LIN {X 0,Y 439.387,Z 629.756,A -85,B 0,C 180,E1 -9133.964,E2 -9133.964} C_VEL
LIN {X 0,Y 439.354,Z 629.76,A -85,B 0,C 180,E1 -9136.541,E2 -9136.541} C_VEL
LIN {X 0,Y 439.382,Z 629.757,A -85,B 0,C 180,E1 -9139.019,E2 -9139.019} C_VEL
LIN {X 0,Y 439.376,Z 629.757,A -85,B 0,C 180,E1 -9141.608,E2 -9141.608} C_VEL
LIN {X 0,Y 439.401,Z 629.753,A -85,B 0,C 180,E1 -9144.844,E2 -9144.844} C_VEL
LIN {X 0,Y 439.375,Z 629.756,A -85,B 0,C 180,E1 -9148.14,E2 -9148.14} C_VEL
LIN {X 0,Y 439.434,Z 629.748,A -85,B 0,C 180,E1 -9151.598,E2 -9151.598} C_VEL
LIN {X 0,Y 439.407,Z 629.752,A -85,B 0,C 180,E1 -9154.415,E2 -9154.415} C_VEL
LIN {X 0,Y 439.367,Z 629.759,A -85,B 0,C 180,E1 -9157.425,E2 -9157.425} C_VEL
LIN {X 0,Y 439.443,Z 629.749,A -85,B 0,C 180,E1 -9160.663,E2 -9160.663} C_VEL
LIN {X 0,Y 439.464,Z 629.745,A -85,B 0,C 180,E1 -9164.225,E2 -9164.225} C_VEL
LIN {X 0,Y 439.485,Z 629.743,A -85,B 0,C 180,E1 -9168.001,E2 -9168.001} C_VEL
LIN {X 0,Y 439.55,Z 629.734,A -85,B 0,C 180,E1 -9171.726,E2 -9171.726} C_VEL
LIN {X 0,Y 439.622,Z 629.725,A -85,B 0,C 180,E1 -9174.496,E2 -9174.496} C_VEL
LIN {X 0,Y 439.636,Z 629.724,A -85,B 0,C 180,E1 -9178.168,E2 -9178.168} C_VEL
LIN {X 0,Y 439.765,Z 629.708,A -85,B 0,C 180,E1 -9180,E2 -9180} C_VEL
LIN {X 0,Y 439.658,Z 629.723,A -85,B 0,C 180,E1 -9182.749,E2 -9182.749} C_VEL
LIN {X 0,Y 439.619,Z 629.727,A -85,B 0,C 180,E1 -9186.425,E2 -9186.425} C_VEL
LIN {X 0,Y 439.538,Z 629.738,A -85,B 0,C 180,E1 -9188.274,E2 -9188.274} C_VEL
LIN {X 0,Y 439.466,Z 630.156,A -85,B 0,C 180,E1 -9189.202,E2 -9189.202} C_VEL
LIN {X 0,Y 439.385,Z 633.62,A -85,B 0,C 180,E1 -9192.002,E2 -9192.002} C_VEL
LIN {X 0,Y 439.192,Z 637.24,A -85,B 0,C 180,E1 -9194.835,E2 -9194.835} C_VEL
LIN {X 0,Y 439.017,Z 641.048,A -85,B 0,C 180,E1 -9197.708,E2 -9197.708} C_VEL
LIN {X 0,Y 438.863,Z 644.989,A -85,B 0,C 180,E1 -9200.629,E2 -9200.629} C_VEL
LIN {X 0,Y 438.726,Z 649.729,A -85,B 0,C 180,E1 -9204.064,E2 -9204.064} C_VEL
LIN {X 0,Y 438.588,Z 653.399,A -85,B 0,C 180,E1 -9206.659,E2 -9206.659} C_VEL
LIN {X 0,Y 438.511,Z 656.226,A -85,B 0,C 180,E1 -9208.638,E2 -9208.638} C_VEL
LIN {X 0,Y 441.656,Z 670.395,A -85,B 0,C 180,E1 -9209.231,E2 -9209.231} C_VEL
LIN {X 0,Y 442.692,Z 676.663,A -85,B 0,C 180,E1 -9209.547,E2 -9209.547} C_VEL
LIN {X 0,Y 442.223,Z 688.254,A -85,B 0,C 180,E1 -9210.172,E2 -9210.172} C_VEL
LIN {X 0,Y 441.639,Z 698.968,A -85,B 0,C 180,E1 -9210.92,E2 -9210.92} C_VEL
LIN {X 0,Y 441.047,Z 709.711,A -85,B 0,C 180,E1 -9211.866,E2 -9211.866} C_VEL
LIN {X 0,Y 440.374,Z 720.086,A -85,B 0,C 180,E1 -9212.998,E2 -9212.998} C_VEL
LIN {X 0,Y 439.839,Z 729.502,A -85,B 0,C 180,E1 -9214.281,E2 -9214.281} C_VEL
LIN {X 0,Y 439.34,Z 736.948,A -85,B 0,C 180,E1 -9215.528,E2 -9215.528} C_VEL
LIN {X 0,Y 438.88,Z 744.552,A -85,B 0,C 180,E1 -9217.12,E2 -9217.12} C_VEL
LIN {X 0,Y 438.615,Z 750.268,A -85,B 0,C 180,E1 -9218.675,E2 -9218.675} C_VEL
LIN {X 0,Y 438.473,Z 753.709,A -85,B 0,C 180,E1 -9219.877,E2 -9219.877} C_VEL
LIN {X 0,Y 438.363,Z 756.384,A -85,B 0,C 180,E1 -9221.103,E2 -9221.103} C_VEL
LIN {X 0,Y 438.248,Z 758.479,A -85,B 0,C 180,E1 -9222.465,E2 -9222.465} C_VEL
LIN {X 0,Y 438.176,Z 759.668,A -85,B 0,C 180,E1 -9223.799,E2 -9223.799} C_VEL
LIN {X 0,Y 438.175,Z 760.031,A -85,B 0,C 180,E1 -9225.111,E2 -9225.111} C_VEL
LIN {X 0,Y 438.146,Z 759.584,A -85,B 0,C 180,E1 -9226.391,E2 -9226.391} C_VEL
LIN {X 0,Y 438.226,Z 758.373,A -85,B 0,C 180,E1 -9227.657,E2 -9227.657} C_VEL
LIN {X 0,Y 438.397,Z 755.222,A -85,B 0,C 180,E1 -9229.514,E2 -9229.514} C_VEL
LIN {X 0,Y 438.527,Z 751.961,A -85,B 0,C 180,E1 -9230.81,E2 -9230.81} C_VEL
LIN {X 0,Y 438.792,Z 746.189,A -85,B 0,C 180,E1 -9232.509,E2 -9232.509} C_VEL
LIN {X 0,Y 439.101,Z 739.867,A -85,B 0,C 180,E1 -9233.945,E2 -9233.945} C_VEL
LIN {X 0,Y 439.519,Z 733.401,A -85,B 0,C 180,E1 -9235.134,E2 -9235.134} C_VEL
LIN {X 0,Y 440.041,Z 725.26,A -85,B 0,C 180,E1 -9236.371,E2 -9236.371} C_VEL
LIN {X 0,Y 440.542,Z 716.573,A -85,B 0,C 180,E1 -9237.457,E2 -9237.457} C_VEL
LIN {X 0,Y 441.236,Z 705.818,A -85,B 0,C 180,E1 -9238.54,E2 -9238.54} C_VEL
LIN {X 0,Y 441.75,Z 695.303,A -85,B 0,C 180,E1 -9239.396,E2 -9239.396} C_VEL
LIN {X 0,Y 442.363,Z 683.212,A -85,B 0,C 180,E1 -9240.167,E2 -9240.167} C_VEL
LIN {X 0,Y 442.46,Z 675.311,A -85,B 0,C 180,E1 -9240.567,E2 -9240.567} C_VEL
LIN {X 0,Y 440.025,Z 662.861,A -85,B 0,C 180,E1 -9241.141,E2 -9241.141} C_VEL
LIN {X 0,Y 438.449,Z 655.721,A -85,B 0,C 180,E1 -9241.42,E2 -9241.42} C_VEL
LIN {X 0,Y 438.576,Z 651.43,A -85,B 0,C 180,E1 -9244.363,E2 -9244.363} C_VEL
LIN {X 0,Y 438.669,Z 647.08,A -85,B 0,C 180,E1 -9247.386,E2 -9247.386} C_VEL
LIN {X 0,Y 438.849,Z 642.879,A -85,B 0,C 180,E1 -9250.348,E2 -9250.348} C_VEL
LIN {X 0,Y 439.018,Z 638.03,A -85,B 0,C 180,E1 -9253.845,E2 -9253.845} C_VEL
LIN {X 0,Y 439.064,Z 636.258,A -85,B 0,C 180,E1 -9255.142,E2 -9255.142} C_VEL
LIN {X 0,Y 438.46,Z 635.313,A -85,B 0,C 180,E1 -9255.899,E2 -9255.899} C_VEL
LIN {X 0,Y 435.671,Z 633.985,A -85,B 0,C 180,E1 -9257.135,E2 -9257.135} C_VEL
LIN {X 0,Y 433.291,Z 632.958,A -85,B 0,C 180,E1 -9258.133,E2 -9258.133} C_VEL
LIN {X 0,Y 432.281,Z 632.076,A -85,B 0,C 180,E1 -9258.902,E2 -9258.902} C_VEL
LIN {X 0,Y 432.206,Z 631.749,A -85,B 0,C 180,E1 -9259.162,E2 -9259.162} C_VEL
LIN {X 0,Y 432.239,Z 631.054,A -85,B 0,C 180,E1 -9259.697,E2 -9259.697} C_VEL
LIN {X 0,Y 432.339,Z 630.633,A -85,B 0,C 180,E1 -9260.644,E2 -9260.644} C_VEL
LIN {X 0,Y 432.557,Z 630.605,A -85,B 0,C 180,E1 -9262.531,E2 -9262.531} C_VEL
LIN {X 0,Y 432.6,Z 630.599,A -85,B 0,C 180,E1 -9264.406,E2 -9264.406} C_VEL
LIN {X 0,Y 432.609,Z 630.596,A -85,B 0,C 180,E1 -9268.138,E2 -9268.138} C_VEL
LIN {X 0,Y 432.738,Z 630.58,A -85,B 0,C 180,E1 -9270,E2 -9270} C_VEL
LIN {X 0,Y 432.608,Z 630.6,A -85,B 0,C 180,E1 -9272.793,E2 -9272.793} C_VEL
LIN {X 0,Y 432.556,Z 630.605,A -85,B 0,C 180,E1 -9276.53,E2 -9276.53} C_VEL
LIN {X 0,Y 432.3,Z 630.637,A -85,B 0,C 180,E1 -9279.356,E2 -9279.356} C_VEL
LIN {X 0,Y 431.893,Z 630.707,A -85,B 0,C 180,E1 -9281.736,E2 -9281.736} C_VEL
LIN {X 0,Y 431.726,Z 636.029,A -85,B 0,C 180,E1 -9285.097,E2 -9285.097} C_VEL
LIN {X 0,Y 431.59,Z 640.656,A -85,B 0,C 180,E1 -9288.022,E2 -9288.022} C_VEL
LIN {X 0,Y 431.486,Z 645.367,A -85,B 0,C 180,E1 -9290.997,E2 -9290.997} C_VEL
LIN {X 0,Y 431.407,Z 650.36,A -85,B 0,C 180,E1 -9294.176,E2 -9294.176} C_VEL
LIN {X 0,Y 431.354,Z 655.502,A -85,B 0,C 180,E1 -9297.437,E2 -9297.437} C_VEL
LIN {X 0,Y 434.318,Z 669.166,A -85,B 0,C 180,E1 -9297.986,E2 -9297.986} C_VEL
LIN {X 0,Y 435.698,Z 677.655,A -85,B 0,C 180,E1 -9298.42,E2 -9298.42} C_VEL
LIN {X 0,Y 435.136,Z 689.502,A -85,B 0,C 180,E1 -9299.085,E2 -9299.085} C_VEL
LIN {X 0,Y 434.575,Z 700.253,A -85,B 0,C 180,E1 -9299.867,E2 -9299.867} C_VEL
LIN {X 0,Y 433.897,Z 711.033,A -85,B 0,C 180,E1 -9300.855,E2 -9300.855} C_VEL
LIN {X 0,Y 433.244,Z 721.833,A -85,B 0,C 180,E1 -9302.09,E2 -9302.09} C_VEL
LIN {X 0,Y 432.678,Z 729.989,A -85,B 0,C 180,E1 -9303.243,E2 -9303.243} C_VEL
LIN {X 0,Y 432.171,Z 738.293,A -85,B 0,C 180,E1 -9304.692,E2 -9304.692} C_VEL
LIN {X 0,Y 431.803,Z 745.011,A -85,B 0,C 180,E1 -9306.157,E2 -9306.157} C_VEL
LIN {X 0,Y 431.499,Z 750.36,A -85,B 0,C 180,E1 -9307.644,E2 -9307.644} C_VEL
LIN {X 0,Y 431.308,Z 754.057,A -85,B 0,C 180,E1 -9308.972,E2 -9308.972} C_VEL
LIN {X 0,Y 431.108,Z 757.46,A -85,B 0,C 180,E1 -9310.698,E2 -9310.698} C_VEL
LIN {X 0,Y 431.064,Z 759.055,A -85,B 0,C 180,E1 -9311.947,E2 -9311.947} C_VEL
LIN {X 0,Y 431.022,Z 759.926,A -85,B 0,C 180,E1 -9313.221,E2 -9313.221} C_VEL
LIN {X 0,Y 431.082,Z 760.032,A -85,B 0,C 180,E1 -9314.509,E2 -9314.509} C_VEL
LIN {X 0,Y 431.091,Z 759.371,A -85,B 0,C 180,E1 -9315.833,E2 -9315.833} C_VEL
LIN {X 0,Y 431.14,Z 757.873,A -85,B 0,C 180,E1 -9317.183,E2 -9317.183} C_VEL
LIN {X 0,Y 431.27,Z 755.46,A -85,B 0,C 180,E1 -9318.556,E2 -9318.556} C_VEL
LIN {X 0,Y 431.458,Z 752.01,A -85,B 0,C 180,E1 -9319.958,E2 -9319.958} C_VEL
LIN {X 0,Y 431.725,Z 747.362,A -85,B 0,C 180,E1 -9321.387,E2 -9321.387} C_VEL
LIN {X 0,Y 432.041,Z 740.614,A -85,B 0,C 180,E1 -9322.995,E2 -9322.995} C_VEL
LIN {X 0,Y 432.534,Z 733.555,A -85,B 0,C 180,E1 -9324.332,E2 -9324.332} C_VEL
LIN {X 0,Y 433.12,Z 724.929,A -85,B 0,C 180,E1 -9325.65,E2 -9325.65} C_VEL
LIN {X 0,Y 433.689,Z 715.93,A -85,B 0,C 180,E1 -9326.773,E2 -9326.773} C_VEL
LIN {X 0,Y 434.381,Z 705.148,A -85,B 0,C 180,E1 -9327.866,E2 -9327.866} C_VEL
LIN {X 0,Y 434.999,Z 694.371,A -85,B 0,C 180,E1 -9328.733,E2 -9328.733} C_VEL
LIN {X 0,Y 435.698,Z 681.528,A -85,B 0,C 180,E1 -9329.53,E2 -9329.53} C_VEL
LIN {X 0,Y 435.721,Z 676.839,A -85,B 0,C 180,E1 -9329.772,E2 -9329.772} C_VEL
LIN {X 0,Y 433.464,Z 664.933,A -85,B 0,C 180,E1 -9330.362,E2 -9330.362} C_VEL
LIN {X 0,Y 431.371,Z 655.826,A -85,B 0,C 180,E1 -9330.74,E2 -9330.74} C_VEL
LIN {X 0,Y 431.529,Z 650.765,A -85,B 0,C 180,E1 -9333.913,E2 -9333.913} C_VEL
LIN {X 0,Y 431.533,Z 645.812,A -85,B 0,C 180,E1 -9336.991,E2 -9336.991} C_VEL
LIN {X 0,Y 431.613,Z 640.991,A -85,B 0,C 180,E1 -9340.004,E2 -9340.004} C_VEL
LIN {X 0,Y 431.703,Z 636.112,A -85,B 0,C 180,E1 -9342.96,E2 -9342.96} C_VEL
LIN {X 0,Y 431.894,Z 630.693,A -85,B 0,C 180,E1 -9346.232,E2 -9346.232} C_VEL
LIN {X 0,Y 432.247,Z 630.647,A -85,B 0,C 180,E1 -9348.749,E2 -9348.749} C_VEL
LIN {X 0,Y 432.486,Z 630.616,A -85,B 0,C 180,E1 -9351.59,E2 -9351.59} C_VEL
LIN {X 0,Y 432.595,Z 630.602,A -85,B 0,C 180,E1 -9354.406,E2 -9354.406} C_VEL
LIN {X 0,Y 432.602,Z 630.601,A -85,B 0,C 180,E1 -9358.138,E2 -9358.138} C_VEL
LIN {X 0,Y 432.731,Z 630.585,A -85,B 0,C 180,E1 -9360,E2 -9360} C_VEL
LIN {X 0,Y 432.603,Z 630.6,A -85,B 0,C 180,E1 -9362.794,E2 -9362.794} C_VEL
LIN {X 0,Y 432.569,Z 630.606,A -85,B 0,C 180,E1 -9366.53,E2 -9366.53} C_VEL
LIN {X 0,Y 432.44,Z 630.621,A -85,B 0,C 180,E1 -9369.353,E2 -9369.353} C_VEL
LIN {X 0,Y 432.427,Z 630.623,A -85,B 0,C 180,E1 -9372.804,E2 -9372.804} C_VEL
LIN {X 0,Y 432.409,Z 630.623,A -85,B 0,C 180,E1 -9376.479,E2 -9376.479} C_VEL
LIN {X 0,Y 432.336,Z 630.634,A -85,B 0,C 180,E1 -9379.961,E2 -9379.961} C_VEL
LIN {X 0,Y 432.316,Z 630.636,A -85,B 0,C 180,E1 -9382.964,E2 -9382.964} C_VEL
LIN {X 0,Y 432.361,Z 630.629,A -85,B 0,C 180,E1 -9386.033,E2 -9386.033} C_VEL
LIN {X 0,Y 432.349,Z 630.632,A -85,B 0,C 180,E1 -9389.187,E2 -9389.187} C_VEL
LIN {X 0,Y 432.323,Z 630.636,A -85,B 0,C 180,E1 -9392.294,E2 -9392.294} C_VEL
LIN {X 0,Y 432.338,Z 630.633,A -85,B 0,C 180,E1 -9394.677,E2 -9394.677} C_VEL
LIN {X 0,Y 432.344,Z 630.631,A -85,B 0,C 180,E1 -9398.149,E2 -9398.149} C_VEL
LIN {X 0,Y 432.33,Z 630.633,A -85,B 0,C 180,E1 -9401.603,E2 -9401.603} C_VEL
LIN {X 0,Y 432.331,Z 630.634,A -85,B 0,C 180,E1 -9404.348,E2 -9404.348} C_VEL
LIN {X 0,Y 432.318,Z 630.636,A -85,B 0,C 180,E1 -9407.016,E2 -9407.016} C_VEL
LIN {X 0,Y 432.41,Z 630.692,A -85,B 0,C 180,E1 -9409.809,E2 -9409.809} C_VEL
LIN {X 0,Y 433.314,Z 636.64,A -85,B 0,C 180,E1 -9413.123,E2 -9413.123} C_VEL
LIN {X 0,Y 433.487,Z 641.023,A -85,B 0,C 180,E1 -9415.428,E2 -9415.428} C_VEL
LIN {X 0,Y 433.031,Z 647.602,A -85,B 0,C 180,E1 -9418.712,E2 -9418.712} C_VEL
LIN {X 0,Y 432.656,Z 654.182,A -85,B 0,C 180,E1 -9421.897,E2 -9421.897} C_VEL
LIN {X 0,Y 432.346,Z 660.779,A -85,B 0,C 180,E1 -9424.999,E2 -9424.999} C_VEL
LIN {X 0,Y 432.028,Z 668.48,A -85,B 0,C 180,E1 -9428.53,E2 -9428.53} C_VEL
LIN {X 0,Y 431.751,Z 675.089,A -85,B 0,C 180,E1 -9431.494,E2 -9431.494} C_VEL
LIN {X 0,Y 431.697,Z 679.324,A -85,B 0,C 180,E1 -9433.355,E2 -9433.355} C_VEL
LIN {X 0,Y 433.966,Z 692.719,A -85,B 0,C 180,E1 -9433.836,E2 -9433.836} C_VEL
LIN {X 0,Y 435.473,Z 703.788,A -85,B 0,C 180,E1 -9434.377,E2 -9434.377} C_VEL
LIN {X 0,Y 434.819,Z 716.766,A -85,B 0,C 180,E1 -9435.133,E2 -9435.133} C_VEL
LIN {X 0,Y 434.143,Z 728.744,A -85,B 0,C 180,E1 -9436.048,E2 -9436.048} C_VEL
LIN {X 0,Y 433.519,Z 739.723,A -85,B 0,C 180,E1 -9437.121,E2 -9437.121} C_VEL
LIN {X 0,Y 432.898,Z 749.427,A -85,B 0,C 180,E1 -9438.292,E2 -9438.292} C_VEL
LIN {X 0,Y 432.369,Z 757.388,A -85,B 0,C 180,E1 -9439.464,E2 -9439.464} C_VEL
LIN {X 0,Y 431.913,Z 765.179,A -85,B 0,C 180,E1 -9440.872,E2 -9440.872} C_VEL
LIN {X 0,Y 431.527,Z 772.331,A -85,B 0,C 180,E1 -9442.514,E2 -9442.514} C_VEL
LIN {X 0,Y 431.315,Z 777.274,A -85,B 0,C 180,E1 -9443.98,E2 -9443.98} C_VEL
LIN {X 0,Y 431.283,Z 780.734,A -85,B 0,C 180,E1 -9445.327,E2 -9445.327} C_VEL
LIN {X 0,Y 431.193,Z 782.61,A -85,B 0,C 180,E1 -9446.262,E2 -9446.262} C_VEL
LIN {X 0,Y 431.228,Z 784.02,A -85,B 0,C 180,E1 -9447.198,E2 -9447.198} C_VEL
LIN {X 0,Y 431.199,Z 785.019,A -85,B 0,C 180,E1 -9448.132,E2 -9448.132} C_VEL
LIN {X 0,Y 431.168,Z 785.627,A -85,B 0,C 180,E1 -9449.066,E2 -9449.066} C_VEL
LIN {X 0,Y 431.167,Z 785.842,A -85,B 0,C 180,E1 -9450,E2 -9450} C_VEL
LIN {X 0,Y 431.168,Z 785.62,A -85,B 0,C 180,E1 -9450.934,E2 -9450.934} C_VEL
LIN {X 0,Y 431.199,Z 785.002,A -85,B 0,C 180,E1 -9451.868,E2 -9451.868} C_VEL
LIN {X 0,Y 431.228,Z 783.992,A -85,B 0,C 180,E1 -9452.803,E2 -9452.803} C_VEL
LIN {X 0,Y 431.193,Z 782.577,A -85,B 0,C 180,E1 -9453.738,E2 -9453.738} C_VEL
LIN {X 0,Y 431.316,Z 779.61,A -85,B 0,C 180,E1 -9455.142,E2 -9455.142} C_VEL
LIN {X 0,Y 431.439,Z 775.597,A -85,B 0,C 180,E1 -9456.548,E2 -9456.548} C_VEL
LIN {X 0,Y 431.685,Z 769.429,A -85,B 0,C 180,E1 -9458.19,E2 -9458.19} C_VEL
LIN {X 0,Y 432.03,Z 762.699,A -85,B 0,C 180,E1 -9459.599,E2 -9459.599} C_VEL
LIN {X 0,Y 432.536,Z 754.358,A -85,B 0,C 180,E1 -9461.007,E2 -9461.007} C_VEL
LIN {X 0,Y 433.169,Z 745.811,A -85,B 0,C 180,E1 -9462.177,E2 -9462.177} C_VEL
LIN {X 0,Y 433.695,Z 736.144,A -85,B 0,C 180,E1 -9463.263,E2 -9463.263} C_VEL
LIN {X 0,Y 434.345,Z 724.87,A -85,B 0,C 180,E1 -9464.286,E2 -9464.286} C_VEL
LIN {X 0,Y 435.053,Z 713.507,A -85,B 0,C 180,E1 -9465.099,E2 -9465.099} C_VEL
LIN {X 0,Y 435.436,Z 703.108,A -85,B 0,C 180,E1 -9465.685,E2 -9465.685} C_VEL
LIN {X 0,Y 433.628,Z 689.975,A -85,B 0,C 180,E1 -9466.313,E2 -9466.313} C_VEL
LIN {X 0,Y 431.674,Z 678.73,A -85,B 0,C 180,E1 -9466.737,E2 -9466.737} C_VEL
LIN {X 0,Y 431.916,Z 670.304,A -85,B 0,C 180,E1 -9470.478,E2 -9470.478} C_VEL
LIN {X 0,Y 432.117,Z 663.72,A -85,B 0,C 180,E1 -9473.483,E2 -9473.483} C_VEL
LIN {X 0,Y 432.477,Z 656.969,A -85,B 0,C 180,E1 -9476.647,E2 -9476.647} C_VEL
LIN {X 0,Y 432.876,Z 649.649,A -85,B 0,C 180,E1 -9480.219,E2 -9480.219} C_VEL
LIN {X 0,Y 433.312,Z 643.31,A -85,B 0,C 180,E1 -9483.467,E2 -9483.467} C_VEL
LIN {X 0,Y 433.508,Z 638.901,A -85,B 0,C 180,E1 -9485.845,E2 -9485.845} C_VEL
LIN {X 0,Y 433.084,Z 635.068,A -85,B 0,C 180,E1 -9488.073,E2 -9488.073} C_VEL
LIN {X 0,Y 432.38,Z 630.631,A -85,B 0,C 180,E1 -9490.862,E2 -9490.862} C_VEL
LIN {X 0,Y 432.343,Z 630.634,A -85,B 0,C 180,E1 -9494.346,E2 -9494.346} C_VEL
LIN {X 0,Y 432.322,Z 630.636,A -85,B 0,C 180,E1 -9497.016,E2 -9497.016} C_VEL
LIN {X 0,Y 432.338,Z 630.635,A -85,B 0,C 180,E1 -9499.82,E2 -9499.82} C_VEL
LIN {X 0,Y 432.308,Z 630.637,A -85,B 0,C 180,E1 -9503.022,E2 -9503.022} C_VEL
LIN {X 0,Y 432.361,Z 630.629,A -85,B 0,C 180,E1 -9505.996,E2 -9505.996} C_VEL
LIN {X 0,Y 432.349,Z 630.631,A -85,B 0,C 180,E1 -9509.49,E2 -9509.49} C_VEL
LIN {X 0,Y 432.393,Z 630.626,A -85,B 0,C 180,E1 -9512.928,E2 -9512.928} C_VEL
LIN {X 0,Y 432.373,Z 630.626,A -85,B 0,C 180,E1 -9516.023,E2 -9516.023} C_VEL
LIN {X 0,Y 432.352,Z 630.631,A -85,B 0,C 180,E1 -9519.046,E2 -9519.046} C_VEL
LIN {X 0,Y 432.38,Z 630.628,A -85,B 0,C 180,E1 -9522.011,E2 -9522.011} C_VEL
LIN {X 0,Y 432.397,Z 630.626,A -85,B 0,C 180,E1 -9524.927,E2 -9524.927} C_VEL
LIN {X 0,Y 432.461,Z 630.619,A -85,B 0,C 180,E1 -9527.803,E2 -9527.803} C_VEL
LIN {X 0,Y 432.494,Z 630.614,A -85,B 0,C 180,E1 -9531.59,E2 -9531.59} C_VEL
LIN {X 0,Y 432.599,Z 630.599,A -85,B 0,C 180,E1 -9534.406,E2 -9534.406} C_VEL
LIN {X 0,Y 432.606,Z 630.6,A -85,B 0,C 180,E1 -9538.138,E2 -9538.138} C_VEL
LIN {X 0,Y 432.735,Z 630.584,A -85,B 0,C 180,E1 -9540,E2 -9540} C_VEL
LIN {X 0,Y 432.607,Z 630.601,A -85,B 0,C 180,E1 -9542.794,E2 -9542.794} C_VEL
LIN {X 0,Y 432.574,Z 630.604,A -85,B 0,C 180,E1 -9546.53,E2 -9546.53} C_VEL
LIN {X 0,Y 432.482,Z 630.617,A -85,B 0,C 180,E1 -9548.41,E2 -9548.41} C_VEL
LIN {X 0,Y 432.441,Z 632.519,A -85,B 0,C 180,E1 -9550.298,E2 -9550.298} C_VEL
LIN {X 0,Y 432.234,Z 636.045,A -85,B 0,C 180,E1 -9553.158,E2 -9553.158} C_VEL
LIN {X 0,Y 432.06,Z 640.081,A -85,B 0,C 180,E1 -9556.319,E2 -9556.319} C_VEL
LIN {X 0,Y 431.934,Z 644.029,A -85,B 0,C 180,E1 -9559.314,E2 -9559.314} C_VEL
LIN {X 0,Y 431.672,Z 649.01,A -85,B 0,C 180,E1 -9563.001,E2 -9563.001} C_VEL
LIN {X 0,Y 431.573,Z 653.721,A -85,B 0,C 180,E1 -9566.407,E2 -9566.407} C_VEL
LIN {X 0,Y 431.451,Z 656.452,A -85,B 0,C 180,E1 -9568.348,E2 -9568.348} C_VEL
LIN {X 0,Y 434.724,Z 671.075,A -85,B 0,C 180,E1 -9568.983,E2 -9568.983} C_VEL
LIN {X 0,Y 435.849,Z 678.398,A -85,B 0,C 180,E1 -9569.364,E2 -9569.364} C_VEL
LIN {X 0,Y 435.193,Z 691.24,A -85,B 0,C 180,E1 -9570.108,E2 -9570.108} C_VEL
LIN {X 0,Y 434.561,Z 702.998,A -85,B 0,C 180,E1 -9571.002,E2 -9571.002} C_VEL
LIN {X 0,Y 433.877,Z 713.737,A -85,B 0,C 180,E1 -9572.039,E2 -9572.039} C_VEL
LIN {X 0,Y 433.224,Z 723.639,A -85,B 0,C 180,E1 -9573.228,E2 -9573.228} C_VEL
LIN {X 0,Y 432.747,Z 731.224,A -85,B 0,C 180,E1 -9574.338,E2 -9574.338} C_VEL
LIN {X 0,Y 432.248,Z 738.456,A -85,B 0,C 180,E1 -9575.614,E2 -9575.614} C_VEL
LIN {X 0,Y 431.806,Z 745.281,A -85,B 0,C 180,E1 -9577.106,E2 -9577.106} C_VEL
LIN {X 0,Y 431.559,Z 750.546,A -85,B 0,C 180,E1 -9578.585,E2 -9578.585} C_VEL
LIN {X 0,Y 431.372,Z 754.495,A -85,B 0,C 180,E1 -9580.027,E2 -9580.027} C_VEL
LIN {X 0,Y 431.223,Z 757.315,A -85,B 0,C 180,E1 -9581.435,E2 -9581.435} C_VEL
LIN {X 0,Y 431.094,Z 759.491,A -85,B 0,C 180,E1 -9583.213,E2 -9583.213} C_VEL
LIN {X 0,Y 431.084,Z 760.172,A -85,B 0,C 180,E1 -9584.51,E2 -9584.51} C_VEL
LIN {X 0,Y 431.08,Z 760.092,A -85,B 0,C 180,E1 -9585.836,E2 -9585.836} C_VEL
LIN {X 0,Y 431.092,Z 759.158,A -85,B 0,C 180,E1 -9587.191,E2 -9587.191} C_VEL
LIN {X 0,Y 431.201,Z 757.333,A -85,B 0,C 180,E1 -9588.568,E2 -9588.568} C_VEL
LIN {X 0,Y 431.374,Z 754.534,A -85,B 0,C 180,E1 -9589.972,E2 -9589.972} C_VEL
LIN {X 0,Y 431.531,Z 750.587,A -85,B 0,C 180,E1 -9591.42,E2 -9591.42} C_VEL
LIN {X 0,Y 431.824,Z 745.029,A -85,B 0,C 180,E1 -9592.974,E2 -9592.974} C_VEL
LIN {X 0,Y 432.181,Z 738.493,A -85,B 0,C 180,E1 -9594.399,E2 -9594.399} C_VEL
LIN {X 0,Y 432.748,Z 729.711,A -85,B 0,C 180,E1 -9595.921,E2 -9595.921} C_VEL
LIN {X 0,Y 433.357,Z 720.825,A -85,B 0,C 180,E1 -9597.159,E2 -9597.159} C_VEL
LIN {X 0,Y 433.943,Z 711.272,A -85,B 0,C 180,E1 -9598.24,E2 -9598.24} C_VEL
LIN {X 0,Y 434.627,Z 699.706,A -85,B 0,C 180,E1 -9599.292,E2 -9599.292} C_VEL
LIN {X 0,Y 435.247,Z 688.292,A -85,B 0,C 180,E1 -9600.109,E2 -9600.109} C_VEL
LIN {X 0,Y 435.644,Z 676.629,A -85,B 0,C 180,E1 -9600.751,E2 -9600.751} C_VEL
LIN {X 0,Y 433.236,Z 664.202,A -85,B 0,C 180,E1 -9601.35,E2 -9601.35} C_VEL
LIN {X 0,Y 431.401,Z 655.914,A -85,B 0,C 180,E1 -9601.689,E2 -9601.689} C_VEL
LIN {X 0,Y 431.5,Z 651.224,A -85,B 0,C 180,E1 -9604.946,E2 -9604.946} C_VEL
LIN {X 0,Y 431.652,Z 646.702,A -85,B 0,C 180,E1 -9608.134,E2 -9608.134} C_VEL
LIN {X 0,Y 431.798,Z 642.711,A -85,B 0,C 180,E1 -9611.002,E2 -9611.002} C_VEL
LIN {X 0,Y 431.965,Z 638.68,A -85,B 0,C 180,E1 -9613.943,E2 -9613.943} C_VEL
LIN {X 0,Y 432.191,Z 634.134,A -85,B 0,C 180,E1 -9617.339,E2 -9617.339} C_VEL
LIN {X 0,Y 432.206,Z 631.749,A -85,B 0,C 180,E1 -9619.162,E2 -9619.162} C_VEL
LIN {X 0,Y 431.584,Z 631.102,A -85,B 0,C 180,E1 -9619.934,E2 -9619.934} C_VEL
LIN {X 0,Y 428.862,Z 631.066,A -85,B 0,C 180,E1 -9621.202,E2 -9621.202} C_VEL
LIN {X 0,Y 426.562,Z 631.349,A -85,B 0,C 180,E1 -9622.23,E2 -9622.23} C_VEL
LIN {X 0,Y 425.595,Z 631.473,A -85,B 0,C 180,E1 -9623.023,E2 -9623.023} C_VEL
LIN {X 0,Y 425.527,Z 631.48,A -85,B 0,C 180,E1 -9623.291,E2 -9623.291} C_VEL
LIN {X 0,Y 425.371,Z 631.5,A -85,B 0,C 180,E1 -9625.261,E2 -9625.261} C_VEL
LIN {X 0,Y 425.579,Z 631.471,A -85,B 0,C 180,E1 -9628.107,E2 -9628.107} C_VEL
LIN {X 0,Y 425.707,Z 631.456,A -85,B 0,C 180,E1 -9630,E2 -9630} C_VEL
LIN {X 0,Y 425.559,Z 631.478,A -85,B 0,C 180,E1 -9632.839,E2 -9632.839} C_VEL
LIN {X 0,Y 425.55,Z 631.475,A -85,B 0,C 180,E1 -9635.686,E2 -9635.686} C_VEL
LIN {X 0,Y 425.343,Z 631.504,A -85,B 0,C 180,E1 -9638.552,E2 -9638.552} C_VEL
LIN {X 0,Y 424.936,Z 631.556,A -85,B 0,C 180,E1 -9641.447,E2 -9641.447} C_VEL
LIN {X 0,Y 424.83,Z 631.781,A -85,B 0,C 180,E1 -9641.934,E2 -9641.934} C_VEL
LIN {X 0,Y 424.662,Z 637.169,A -85,B 0,C 180,E1 -9645.354,E2 -9645.354} C_VEL
LIN {X 0,Y 424.515,Z 641.84,A -85,B 0,C 180,E1 -9648.333,E2 -9648.333} C_VEL
LIN {X 0,Y 424.414,Z 647.522,A -85,B 0,C 180,E1 -9651.978,E2 -9651.978} C_VEL
LIN {X 0,Y 424.292,Z 653.067,A -85,B 0,C 180,E1 -9655.509,E2 -9655.509} C_VEL
LIN {X 0,Y 424.269,Z 655.655,A -85,B 0,C 180,E1 -9657.165,E2 -9657.165} C_VEL
LIN {X 0,Y 427.366,Z 669.765,A -85,B 0,C 180,E1 -9657.748,E2 -9657.748} C_VEL
LIN {X 0,Y 428.784,Z 677.926,A -85,B 0,C 180,E1 -9658.18,E2 -9658.18} C_VEL
LIN {X 0,Y 428.249,Z 690.213,A -85,B 0,C 180,E1 -9658.887,E2 -9658.887} C_VEL
LIN {X 0,Y 427.658,Z 700.736,A -85,B 0,C 180,E1 -9659.673,E2 -9659.673} C_VEL
LIN {X 0,Y 426.933,Z 711.53,A -85,B 0,C 180,E1 -9660.684,E2 -9660.684} C_VEL
LIN {X 0,Y 426.292,Z 721.503,A -85,B 0,C 180,E1 -9661.84,E2 -9661.84} C_VEL
LIN {X 0,Y 425.713,Z 729.756,A -85,B 0,C 180,E1 -9663.01,E2 -9663.01} C_VEL
LIN {X 0,Y 425.152,Z 738.171,A -85,B 0,C 180,E1 -9664.488,E2 -9664.488} C_VEL
LIN {X 0,Y 424.786,Z 744.361,A -85,B 0,C 180,E1 -9665.836,E2 -9665.836} C_VEL
LIN {X 0,Y 424.454,Z 749.97,A -85,B 0,C 180,E1 -9667.366,E2 -9667.366} C_VEL
LIN {X 0,Y 424.213,Z 754.514,A -85,B 0,C 180,E1 -9669.016,E2 -9669.016} C_VEL
LIN {X 0,Y 424.037,Z 757.147,A -85,B 0,C 180,E1 -9670.323,E2 -9670.323} C_VEL
LIN {X 0,Y 423.972,Z 759.096,A -85,B 0,C 180,E1 -9671.759,E2 -9671.759} C_VEL
LIN {X 0,Y 423.924,Z 760.093,A -85,B 0,C 180,E1 -9673.159,E2 -9673.159} C_VEL
LIN {X 0,Y 423.984,Z 760.228,A -85,B 0,C 180,E1 -9674.539,E2 -9674.539} C_VEL
LIN {X 0,Y 423.994,Z 759.564,A -85,B 0,C 180,E1 -9675.878,E2 -9675.878} C_VEL
LIN {X 0,Y 424.046,Z 758.147,A -85,B 0,C 180,E1 -9677.194,E2 -9677.194} C_VEL
LIN {X 0,Y 424.18,Z 755.971,A -85,B 0,C 180,E1 -9678.491,E2 -9678.491} C_VEL
LIN {X 0,Y 424.352,Z 753.007,A -85,B 0,C 180,E1 -9679.766,E2 -9679.766} C_VEL
LIN {X 0,Y 424.634,Z 748.084,A -85,B 0,C 180,E1 -9681.375,E2 -9681.375} C_VEL
LIN {X 0,Y 424.997,Z 741.412,A -85,B 0,C 180,E1 -9683.019,E2 -9683.019} C_VEL
LIN {X 0,Y 425.494,Z 734.476,A -85,B 0,C 180,E1 -9684.378,E2 -9684.378} C_VEL
LIN {X 0,Y 426.106,Z 725.939,A -85,B 0,C 180,E1 -9685.736,E2 -9685.736} C_VEL
LIN {X 0,Y 426.728,Z 716.57,A -85,B 0,C 180,E1 -9686.937,E2 -9686.937} C_VEL
LIN {X 0,Y 427.448,Z 706.609,A -85,B 0,C 180,E1 -9687.978,E2 -9687.978} C_VEL
LIN {X 0,Y 428.096,Z 695.689,A -85,B 0,C 180,E1 -9688.9,E2 -9688.9} C_VEL
LIN {X 0,Y 428.767,Z 683.987,A -85,B 0,C 180,E1 -9689.665,E2 -9689.665} C_VEL
LIN {X 0,Y 428.856,Z 677.61,A -85,B 0,C 180,E1 -9690.011,E2 -9690.011} C_VEL
LIN {X 0,Y 426.364,Z 664.772,A -85,B 0,C 180,E1 -9690.668,E2 -9690.668} C_VEL
LIN {X 0,Y 424.308,Z 656.041,A -85,B 0,C 180,E1 -9691.021,E2 -9691.021} C_VEL
LIN {X 0,Y 424.436,Z 650.526,A -85,B 0,C 180,E1 -9694.499,E2 -9694.499} C_VEL
LIN {X 0,Y 424.502,Z 644.97,A -85,B 0,C 180,E1 -9697.99,E2 -9697.99} C_VEL
LIN {X 0,Y 424.619,Z 640.631,A -85,B 0,C 180,E1 -9700.669,E2 -9700.669} C_VEL
LIN {X 0,Y 424.69,Z 635.637,A -85,B 0,C 180,E1 -9703.699,E2 -9703.699} C_VEL
LIN {X 0,Y 424.852,Z 631.57,A -85,B 0,C 180,E1 -9706.121,E2 -9706.121} C_VEL
LIN {X 0,Y 425.187,Z 631.526,A -85,B 0,C 180,E1 -9708.559,E2 -9708.559} C_VEL
LIN {X 0,Y 425.435,Z 631.495,A -85,B 0,C 180,E1 -9711.45,E2 -9711.45} C_VEL
LIN {X 0,Y 425.551,Z 631.48,A -85,B 0,C 180,E1 -9714.313,E2 -9714.313} C_VEL
LIN {X 0,Y 425.572,Z 631.477,A -85,B 0,C 180,E1 -9718.107,E2 -9718.107} C_VEL
LIN {X 0,Y 425.701,Z 631.46,A -85,B 0,C 180,E1 -9720,E2 -9720} C_VEL
LIN {X 0,Y 425.554,Z 631.478,A -85,B 0,C 180,E1 -9722.84,E2 -9722.84} C_VEL
LIN {X 0,Y 425.527,Z 631.482,A -85,B 0,C 180,E1 -9726.639,E2 -9726.639} C_VEL
LIN {X 0,Y 425.399,Z 631.497,A -85,B 0,C 180,E1 -9729.509,E2 -9729.509} C_VEL
LIN {X 0,Y 425.389,Z 631.499,A -85,B 0,C 180,E1 -9732.904,E2 -9732.904} C_VEL
LIN {X 0,Y 425.358,Z 631.502,A -85,B 0,C 180,E1 -9736.605,E2 -9736.605} C_VEL
LIN {X 0,Y 425.325,Z 631.506,A -85,B 0,C 180,E1 -9739.636,E2 -9739.636} C_VEL
LIN {X 0,Y 425.303,Z 631.508,A -85,B 0,C 180,E1 -9743.365,E2 -9743.365} C_VEL
LIN {X 0,Y 425.345,Z 631.503,A -85,B 0,C 180,E1 -9746.845,E2 -9746.845} C_VEL
LIN {X 0,Y 425.315,Z 631.508,A -85,B 0,C 180,E1 -9749.718,E2 -9749.718} C_VEL
LIN {X 0,Y 425.279,Z 631.512,A -85,B 0,C 180,E1 -9753.048,E2 -9753.048} C_VEL
LIN {X 0,Y 425.282,Z 631.511,A -85,B 0,C 180,E1 -9755.93,E2 -9755.93} C_VEL
LIN {X 0,Y 425.298,Z 631.51,A -85,B 0,C 180,E1 -9759.044,E2 -9759.044} C_VEL
LIN {X 0,Y 425.272,Z 631.514,A -85,B 0,C 180,E1 -9762.654,E2 -9762.654} C_VEL
LIN {X 0,Y 425.259,Z 631.515,A -85,B 0,C 180,E1 -9766.045,E2 -9766.045} C_VEL
LIN {X 0,Y 425.319,Z 631.515,A -85,B 0,C 180,E1 -9769.553,E2 -9769.553} C_VEL
LIN {X 0,Y 426.135,Z 636.492,A -85,B 0,C 180,E1 -9772.395,E2 -9772.395} C_VEL
LIN {X 0,Y 426.51,Z 640.877,A -85,B 0,C 180,E1 -9774.78,E2 -9774.78} C_VEL
LIN {X 0,Y 426.085,Z 647.443,A -85,B 0,C 180,E1 -9778.142,E2 -9778.142} C_VEL
LIN {X 0,Y 425.693,Z 654.008,A -85,B 0,C 180,E1 -9781.395,E2 -9781.395} C_VEL
LIN {X 0,Y 425.318,Z 660.596,A -85,B 0,C 180,E1 -9784.557,E2 -9784.557} C_VEL
LIN {X 0,Y 425.031,Z 667.563,A -85,B 0,C 180,E1 -9787.816,E2 -9787.816} C_VEL
LIN {X 0,Y 424.698,Z 674.878,A -85,B 0,C 180,E1 -9791.175,E2 -9791.175} C_VEL
LIN {X 0,Y 424.626,Z 679.046,A -85,B 0,C 180,E1 -9793.059,E2 -9793.059} C_VEL
LIN {X 0,Y 427.211,Z 694.635,A -85,B 0,C 180,E1 -9793.671,E2 -9793.671} C_VEL
LIN {X 0,Y 428.515,Z 705.594,A -85,B 0,C 180,E1 -9794.239,E2 -9794.239} C_VEL
LIN {X 0,Y 427.843,Z 718.128,A -85,B 0,C 180,E1 -9795.006,E2 -9795.006} C_VEL
LIN {X 0,Y 427.143,Z 729.533,A -85,B 0,C 180,E1 -9795.921,E2 -9795.921} C_VEL
LIN {X 0,Y 426.483,Z 740.471,A -85,B 0,C 180,E1 -9797.025,E2 -9797.025} C_VEL
LIN {X 0,Y 425.893,Z 749.122,A -85,B 0,C 180,E1 -9798.096,E2 -9798.096} C_VEL
LIN {X 0,Y 425.336,Z 757.1,A -85,B 0,C 180,E1 -9799.288,E2 -9799.288} C_VEL
LIN {X 0,Y 424.858,Z 764.912,A -85,B 0,C 180,E1 -9800.719,E2 -9800.719} C_VEL
LIN {X 0,Y 424.558,Z 770.238,A -85,B 0,C 180,E1 -9801.912,E2 -9801.912} C_VEL
LIN {X 0,Y 424.259,Z 776.436,A -85,B 0,C 180,E1 -9803.681,E2 -9803.681} C_VEL
LIN {X 0,Y 424.213,Z 780.503,A -85,B 0,C 180,E1 -9805.249,E2 -9805.249} C_VEL
LIN {X 0,Y 424.105,Z 782.384,A -85,B 0,C 180,E1 -9806.2,E2 -9806.2} C_VEL
LIN {X 0,Y 424.125,Z 783.799,A -85,B 0,C 180,E1 -9807.151,E2 -9807.151} C_VEL
LIN {X 0,Y 424.125,Z 784.803,A -85,B 0,C 180,E1 -9808.101,E2 -9808.101} C_VEL
LIN {X 0,Y 424.084,Z 785.631,A -85,B 0,C 180,E1 -9810,E2 -9810} C_VEL
LIN {X 0,Y 424.088,Z 785.413,A -85,B 0,C 180,E1 -9810.95,E2 -9810.95} C_VEL
LIN {X 0,Y 424.125,Z 784.797,A -85,B 0,C 180,E1 -9811.9,E2 -9811.9} C_VEL
LIN {X 0,Y 424.125,Z 783.788,A -85,B 0,C 180,E1 -9812.85,E2 -9812.85} C_VEL
LIN {X 0,Y 424.105,Z 782.375,A -85,B 0,C 180,E1 -9813.801,E2 -9813.801} C_VEL
LIN {X 0,Y 424.23,Z 779.409,A -85,B 0,C 180,E1 -9815.228,E2 -9815.228} C_VEL
LIN {X 0,Y 424.354,Z 775.397,A -85,B 0,C 180,E1 -9816.658,E2 -9816.658} C_VEL
LIN {X 0,Y 424.619,Z 769.234,A -85,B 0,C 180,E1 -9818.327,E2 -9818.327} C_VEL
LIN {X 0,Y 425,Z 762.505,A -85,B 0,C 180,E1 -9819.759,E2 -9819.759} C_VEL
LIN {X 0,Y 425.519,Z 754.166,A -85,B 0,C 180,E1 -9821.191,E2 -9821.191} C_VEL
LIN {X 0,Y 426.205,Z 745.627,A -85,B 0,C 180,E1 -9822.379,E2 -9822.379} C_VEL
LIN {X 0,Y 426.812,Z 735.336,A -85,B 0,C 180,E1 -9823.546,E2 -9823.546} C_VEL
LIN {X 0,Y 427.442,Z 724.71,A -85,B 0,C 180,E1 -9824.522,E2 -9824.522} C_VEL
LIN {X 0,Y 428.175,Z 713.391,A -85,B 0,C 180,E1 -9825.348,E2 -9825.348} C_VEL
LIN {X 0,Y 428.571,Z 704.164,A -85,B 0,C 180,E1 -9825.882,E2 -9825.882} C_VEL
LIN {X 0,Y 426.767,Z 690.673,A -85,B 0,C 180,E1 -9826.564,E2 -9826.564} C_VEL
LIN {X 0,Y 424.617,Z 678.562,A -85,B 0,C 180,E1 -9827.02,E2 -9827.02} C_VEL
LIN {X 0,Y 424.889,Z 670.148,A -85,B 0,C 180,E1 -9830.832,E2 -9830.832} C_VEL
LIN {X 0,Y 425.111,Z 663.586,A -85,B 0,C 180,E1 -9833.894,E2 -9833.894} C_VEL
LIN {X 0,Y 425.443,Z 657.379,A -85,B 0,C 180,E1 -9836.869,E2 -9836.869} C_VEL
LIN {X 0,Y 425.842,Z 650.643,A -85,B 0,C 180,E1 -9840.223,E2 -9840.223} C_VEL
LIN {X 0,Y 426.311,Z 644.319,A -85,B 0,C 180,E1 -9843.523,E2 -9843.523} C_VEL
LIN {X 0,Y 426.521,Z 641.219,A -85,B 0,C 180,E1 -9845.22,E2 -9845.22} C_VEL
LIN {X 0,Y 426.201,Z 637.003,A -85,B 0,C 180,E1 -9847.673,E2 -9847.673} C_VEL
LIN {X 0,Y 425.493,Z 632.453,A -85,B 0,C 180,E1 -9850.554,E2 -9850.554} C_VEL
LIN {X 0,Y 425.313,Z 631.511,A -85,B 0,C 180,E1 -9851.261,E2 -9851.261} C_VEL
LIN {X 0,Y 425.291,Z 631.511,A -85,B 0,C 180,E1 -9854.718,E2 -9854.718} C_VEL
LIN {X 0,Y 425.292,Z 631.512,A -85,B 0,C 180,E1 -9858.042,E2 -9858.042} C_VEL
LIN {X 0,Y 425.309,Z 631.511,A -85,B 0,C 180,E1 -9861.102,E2 -9861.102} C_VEL
LIN {X 0,Y 425.301,Z 631.51,A -85,B 0,C 180,E1 -9864.664,E2 -9864.664} C_VEL
LIN {X 0,Y 425.267,Z 631.513,A -85,B 0,C 180,E1 -9868.073,E2 -9868.073} C_VEL
LIN {X 0,Y 425.333,Z 631.505,A -85,B 0,C 180,E1 -9871.368,E2 -9871.368} C_VEL
LIN {X 0,Y 425.297,Z 631.511,A -85,B 0,C 180,E1 -9874.555,E2 -9874.555} C_VEL
LIN {X 0,Y 425.289,Z 631.511,A -85,B 0,C 180,E1 -9877.661,E2 -9877.661} C_VEL
LIN {X 0,Y 425.364,Z 631.503,A -85,B 0,C 180,E1 -9880.704,E2 -9880.704} C_VEL
LIN {X 0,Y 425.39,Z 631.499,A -85,B 0,C 180,E1 -9883.688,E2 -9883.688} C_VEL
LIN {X 0,Y 425.414,Z 631.496,A -85,B 0,C 180,E1 -9887.598,E2 -9887.598} C_VEL
LIN {X 0,Y 425.444,Z 631.493,A -85,B 0,C 180,E1 -9891.45,E2 -9891.45} C_VEL
LIN {X 0,Y 425.556,Z 631.477,A -85,B 0,C 180,E1 -9894.313,E2 -9894.313} C_VEL
LIN {X 0,Y 425.575,Z 631.476,A -85,B 0,C 180,E1 -9898.107,E2 -9898.107} C_VEL
LIN {X 0,Y 425.705,Z 631.46,A -85,B 0,C 180,E1 -9900,E2 -9900} C_VEL
LIN {X 0,Y 425.559,Z 631.479,A -85,B 0,C 180,E1 -9902.84,E2 -9902.84} C_VEL
LIN {X 0,Y 425.531,Z 631.482,A -85,B 0,C 180,E1 -9906.639,E2 -9906.639} C_VEL
LIN {X 0,Y 425.421,Z 631.501,A -85,B 0,C 180,E1 -9908.551,E2 -9908.551} C_VEL
LIN {X 0,Y 425.322,Z 634.917,A -85,B 0,C 180,E1 -9911.437,E2 -9911.437} C_VEL
LIN {X 0,Y 425.126,Z 638.495,A -85,B 0,C 180,E1 -9914.358,E2 -9914.358} C_VEL
LIN {X 0,Y 424.933,Z 642.278,A -85,B 0,C 180,E1 -9917.32,E2 -9917.32} C_VEL
LIN {X 0,Y 424.761,Z 646.215,A -85,B 0,C 180,E1 -9920.332,E2 -9920.332} C_VEL
LIN {X 0,Y 424.597,Z 650.311,A -85,B 0,C 180,E1 -9923.407,E2 -9923.407} C_VEL
LIN {X 0,Y 424.478,Z 654.692,A -85,B 0,C 180,E1 -9926.611,E2 -9926.611} C_VEL
LIN {X 0,Y 424.404,Z 656.887,A -85,B 0,C 180,E1 -9928.06,E2 -9928.06} C_VEL
LIN {X 0,Y 427.424,Z 669.755,A -85,B 0,C 180,E1 -9928.621,E2 -9928.621} C_VEL
LIN {X 0,Y 429.021,Z 678.909,A -85,B 0,C 180,E1 -9929.112,E2 -9929.112} C_VEL
LIN {X 0,Y 428.366,Z 691.633,A -85,B 0,C 180,E1 -9929.867,E2 -9929.867} C_VEL
LIN {X 0,Y 427.736,Z 702.77,A -85,B 0,C 180,E1 -9930.726,E2 -9930.726} C_VEL
LIN {X 0,Y 426.997,Z 713.635,A -85,B 0,C 180,E1 -9931.782,E2 -9931.782} C_VEL
LIN {X 0,Y 426.295,Z 723.361,A -85,B 0,C 180,E1 -9932.96,E2 -9932.96} C_VEL
LIN {X 0,Y 425.681,Z 732.719,A -85,B 0,C 180,E1 -9934.361,E2 -9934.361} C_VEL
LIN {X 0,Y 425.087,Z 740.815,A -85,B 0,C 180,E1 -9935.892,E2 -9935.892} C_VEL
LIN {X 0,Y 424.683,Z 747.155,A -85,B 0,C 180,E1 -9937.407,E2 -9937.407} C_VEL
LIN {X 0,Y 424.434,Z 752.314,A -85,B 0,C 180,E1 -9938.993,E2 -9938.993} C_VEL
LIN {X 0,Y 424.2,Z 756.703,A -85,B 0,C 180,E1 -9940.899,E2 -9940.899} C_VEL
LIN {X 0,Y 424.092,Z 758.15,A -85,B 0,C 180,E1 -9941.778,E2 -9941.778} C_VEL
LIN {X 0,Y 424.001,Z 759.701,A -85,B 0,C 180,E1 -9943.17,E2 -9943.17} C_VEL
LIN {X 0,Y 423.986,Z 760.391,A -85,B 0,C 180,E1 -9944.539,E2 -9944.539} C_VEL
LIN {X 0,Y 423.98,Z 760.285,A -85,B 0,C 180,E1 -9945.877,E2 -9945.877} C_VEL
LIN {X 0,Y 423.995,Z 759.393,A -85,B 0,C 180,E1 -9947.187,E2 -9947.187} C_VEL
LIN {X 0,Y 424.115,Z 757.745,A -85,B 0,C 180,E1 -9948.483,E2 -9948.483} C_VEL
LIN {X 0,Y 424.274,Z 755.383,A -85,B 0,C 180,E1 -9949.757,E2 -9949.757} C_VEL
LIN {X 0,Y 424.405,Z 752.019,A -85,B 0,C 180,E1 -9951.106,E2 -9951.106} C_VEL
LIN {X 0,Y 424.675,Z 747.135,A -85,B 0,C 180,E1 -9952.595,E2 -9952.595} C_VEL
LIN {X 0,Y 425.02,Z 740.734,A -85,B 0,C 180,E1 -9954.121,E2 -9954.121} C_VEL
LIN {X 0,Y 425.558,Z 732.559,A -85,B 0,C 180,E1 -9955.664,E2 -9955.664} C_VEL
LIN {X 0,Y 426.229,Z 723.373,A -85,B 0,C 180,E1 -9957.035,E2 -9957.035} C_VEL
LIN {X 0,Y 426.893,Z 713.677,A -85,B 0,C 180,E1 -9958.209,E2 -9958.209} C_VEL
LIN {X 0,Y 427.574,Z 702.873,A -85,B 0,C 180,E1 -9959.264,E2 -9959.264} C_VEL
LIN {X 0,Y 428.2,Z 691.606,A -85,B 0,C 180,E1 -9960.134,E2 -9960.134} C_VEL
LIN {X 0,Y 428.872,Z 679.153,A -85,B 0,C 180,E1 -9960.874,E2 -9960.874} C_VEL
LIN {X 0,Y 427.154,Z 668.955,A -85,B 0,C 180,E1 -9961.409,E2 -9961.409} C_VEL
LIN {X 0,Y 424.331,Z 656.082,A -85,B 0,C 180,E1 -9961.968,E2 -9961.968} C_VEL
LIN {X 0,Y 424.432,Z 652.486,A -85,B 0,C 180,E1 -9964.499,E2 -9964.499} C_VEL
LIN {X 0,Y 424.578,Z 647.626,A -85,B 0,C 180,E1 -9967.967,E2 -9967.967} C_VEL
LIN {X 0,Y 424.728,Z 643.893,A -85,B 0,C 180,E1 -9970.674,E2 -9970.674} C_VEL
LIN {X 0,Y 424.899,Z 639.838,A -85,B 0,C 180,E1 -9973.669,E2 -9973.669} C_VEL
LIN {X 0,Y 425.154,Z 635.113,A -85,B 0,C 180,E1 -9977.24,E2 -9977.24} C_VEL
LIN {X 0,Y 425.184,Z 632.162,A -85,B 0,C 180,E1 -9979.524,E2 -9979.524} C_VEL
LIN {X 0,Y 425.261,Z 631.514,A -85,B 0,C 180,E1 -9980.487,E2 -9980.487} C_VEL
LIN {X 0,Y 425.541,Z 631.477,A -85,B 0,C 180,E1 -9982.407,E2 -9982.407} C_VEL
LIN {X 0,Y 425.527,Z 631.48,A -85,B 0,C 180,E1 -9983.291,E2 -9983.291} C_VEL
LIN {X 0,Y 424.887,Z 631.565,A -85,B 0,C 180,E1 -9984.079,E2 -9984.079} C_VEL
LIN {X 0,Y 422.038,Z 631.923,A -85,B 0,C 180,E1 -9985.36,E2 -9985.36} C_VEL
LIN {X 0,Y 419.617,Z 632.221,A -85,B 0,C 180,E1 -9986.394,E2 -9986.394} C_VEL
LIN {X 0,Y 418.589,Z 632.345,A -85,B 0,C 180,E1 -9987.193,E2 -9987.193} C_VEL
LIN {X 0,Y 418.512,Z 632.352,A -85,B 0,C 180,E1 -9987.464,E2 -9987.464} C_VEL
LIN {X 0,Y 418.677,Z 632.331,A -85,B 0,C 180,E1 -9990,E2 -9990} C_VEL
LIN {X 0,Y 418.513,Z 632.356,A -85,B 0,C 180,E1 -9992.887,E2 -9992.887} C_VEL
LIN {X 0,Y 418.508,Z 632.352,A -85,B 0,C 180,E1 -9995.782,E2 -9995.782} C_VEL
LIN {X 0,Y 418.271,Z 632.386,A -85,B 0,C 180,E1 -9998.697,E2 -9998.697} C_VEL
LIN {X 0,Y 417.807,Z 632.443,A -85,B 0,C 180,E1 -10001.763,E2 -10001.763} C_VEL
LIN {X 0,Y 417.594,Z 638.307,A -85,B 0,C 180,E1 -10005.621,E2 -10005.621} C_VEL
LIN {X 0,Y 417.459,Z 643.024,A -85,B 0,C 180,E1 -10008.654,E2 -10008.654} C_VEL
LIN {X 0,Y 417.32,Z 648.438,A -85,B 0,C 180,E1 -10012.143,E2 -10012.143} C_VEL
LIN {X 0,Y 417.244,Z 652.723,A -85,B 0,C 180,E1 -10014.903,E2 -10014.903} C_VEL
LIN {X 0,Y 417.221,Z 655.949,A -85,B 0,C 180,E1 -10016.899,E2 -10016.899} C_VEL
LIN {X 0,Y 420.273,Z 669.775,A -85,B 0,C 180,E1 -10017.472,E2 -10017.472} C_VEL
LIN {X 0,Y 421.919,Z 679.749,A -85,B 0,C 180,E1 -10018.014,E2 -10018.014} C_VEL
LIN {X 0,Y 421.273,Z 692.301,A -85,B 0,C 180,E1 -10018.783,E2 -10018.783} C_VEL
LIN {X 0,Y 420.531,Z 704.452,A -85,B 0,C 180,E1 -10019.757,E2 -10019.757} C_VEL
LIN {X 0,Y 419.771,Z 715.11,A -85,B 0,C 180,E1 -10020.846,E2 -10020.846} C_VEL
LIN {X 0,Y 419.028,Z 725.533,A -85,B 0,C 180,E1 -10022.175,E2 -10022.175} C_VEL
LIN {X 0,Y 418.458,Z 733.688,A -85,B 0,C 180,E1 -10023.461,E2 -10023.461} C_VEL
LIN {X 0,Y 417.984,Z 740.899,A -85,B 0,C 180,E1 -10024.867,E2 -10024.867} C_VEL
LIN {X 0,Y 417.585,Z 747.163,A -85,B 0,C 180,E1 -10026.387,E2 -10026.387} C_VEL
LIN {X 0,Y 417.278,Z 752.551,A -85,B 0,C 180,E1 -10028.076,E2 -10028.076} C_VEL
LIN {X 0,Y 417.002,Z 756.527,A -85,B 0,C 180,E1 -10029.824,E2 -10029.824} C_VEL
LIN {X 0,Y 416.887,Z 758.57,A -85,B 0,C 180,E1 -10031.107,E2 -10031.107} C_VEL
LIN {X 0,Y 416.855,Z 759.868,A -85,B 0,C 180,E1 -10032.405,E2 -10032.405} C_VEL
LIN {X 0,Y 416.85,Z 760.44,A -85,B 0,C 180,E1 -10033.728,E2 -10033.728} C_VEL
LIN {X 0,Y 416.892,Z 760.269,A -85,B 0,C 180,E1 -10035.075,E2 -10035.075} C_VEL
LIN {X 0,Y 416.915,Z 759.298,A -85,B 0,C 180,E1 -10036.456,E2 -10036.456} C_VEL
LIN {X 0,Y 417.072,Z 756.498,A -85,B 0,C 180,E1 -10038.394,E2 -10038.394} C_VEL
LIN {X 0,Y 417.261,Z 753.502,A -85,B 0,C 180,E1 -10039.753,E2 -10039.753} C_VEL
LIN {X 0,Y 417.574,Z 748.36,A -85,B 0,C 180,E1 -10041.484,E2 -10041.484} C_VEL
LIN {X 0,Y 417.934,Z 742.344,A -85,B 0,C 180,E1 -10043.016,E2 -10043.016} C_VEL
LIN {X 0,Y 418.506,Z 734.5,A -85,B 0,C 180,E1 -10044.594,E2 -10044.594} C_VEL
LIN {X 0,Y 419.188,Z 725.905,A -85,B 0,C 180,E1 -10045.975,E2 -10045.975} C_VEL
LIN {X 0,Y 419.876,Z 716.265,A -85,B 0,C 180,E1 -10047.223,E2 -10047.223} C_VEL
LIN {X 0,Y 420.602,Z 705.817,A -85,B 0,C 180,E1 -10048.32,E2 -10048.32} C_VEL
LIN {X 0,Y 421.379,Z 694.142,A -85,B 0,C 180,E1 -10049.284,E2 -10049.284} C_VEL
LIN {X 0,Y 422.062,Z 682.514,A -85,B 0,C 180,E1 -10050.03,E2 -10050.03} C_VEL
LIN {X 0,Y 421.907,Z 677.83,A -85,B 0,C 180,E1 -10050.293,E2 -10050.293} C_VEL
LIN {X 0,Y 419.512,Z 665.695,A -85,B 0,C 180,E1 -10050.933,E2 -10050.933} C_VEL
LIN {X 0,Y 417.251,Z 656.186,A -85,B 0,C 180,E1 -10051.348,E2 -10051.348} C_VEL
LIN {X 0,Y 417.346,Z 651.983,A -85,B 0,C 180,E1 -10054.034,E2 -10054.034} C_VEL
LIN {X 0,Y 417.437,Z 645.983,A -85,B 0,C 180,E1 -10057.815,E2 -10057.815} C_VEL
LIN {X 0,Y 417.555,Z 640.394,A -85,B 0,C 180,E1 -10061.349,E2 -10061.349} C_VEL
LIN {X 0,Y 417.676,Z 635.415,A -85,B 0,C 180,E1 -10064.382,E2 -10064.382} C_VEL
LIN {X 0,Y 417.778,Z 632.452,A -85,B 0,C 180,E1 -10066.13,E2 -10066.13} C_VEL
LIN {X 0,Y 418.13,Z 632.405,A -85,B 0,C 180,E1 -10068.364,E2 -10068.364} C_VEL
LIN {X 0,Y 418.391,Z 632.372,A -85,B 0,C 180,E1 -10071.305,E2 -10071.305} C_VEL
LIN {X 0,Y 418.51,Z 632.358,A -85,B 0,C 180,E1 -10074.217,E2 -10074.217} C_VEL
LIN {X 0,Y 418.541,Z 632.352,A -85,B 0,C 180,E1 -10078.075,E2 -10078.075} C_VEL
LIN {X 0,Y 418.671,Z 632.336,A -85,B 0,C 180,E1 -10080,E2 -10080} C_VEL
LIN {X 0,Y 418.508,Z 632.356,A -85,B 0,C 180,E1 -10082.888,E2 -10082.888} C_VEL
LIN {X 0,Y 418.49,Z 632.358,A -85,B 0,C 180,E1 -10086.751,E2 -10086.751} C_VEL
LIN {X 0,Y 418.339,Z 632.376,A -85,B 0,C 180,E1 -10089.671,E2 -10089.671} C_VEL
LIN {X 0,Y 418.342,Z 632.376,A -85,B 0,C 180,E1 -10093.001,E2 -10093.001} C_VEL
LIN {X 0,Y 418.309,Z 632.38,A -85,B 0,C 180,E1 -10096.736,E2 -10096.736} C_VEL
LIN {X 0,Y 418.267,Z 632.386,A -85,B 0,C 180,E1 -10099.791,E2 -10099.791} C_VEL
LIN {X 0,Y 418.234,Z 632.39,A -85,B 0,C 180,E1 -10102.736,E2 -10102.736} C_VEL
LIN {X 0,Y 418.268,Z 632.385,A -85,B 0,C 180,E1 -10105.904,E2 -10105.904} C_VEL
LIN {X 0,Y 418.272,Z 632.385,A -85,B 0,C 180,E1 -10109.162,E2 -10109.162} C_VEL
LIN {X 0,Y 418.255,Z 632.387,A -85,B 0,C 180,E1 -10112.845,E2 -10112.845} C_VEL
LIN {X 0,Y 418.245,Z 632.388,A -85,B 0,C 180,E1 -10116.239,E2 -10116.239} C_VEL
LIN {X 0,Y 418.249,Z 632.386,A -85,B 0,C 180,E1 -10119.682,E2 -10119.682} C_VEL
LIN {X 0,Y 418.227,Z 632.39,A -85,B 0,C 180,E1 -10122.322,E2 -10122.322} C_VEL
LIN {X 0,Y 418.233,Z 632.39,A -85,B 0,C 180,E1 -10125.109,E2 -10125.109} C_VEL
LIN {X 0,Y 418.238,Z 632.39,A -85,B 0,C 180,E1 -10127.767,E2 -10127.767} C_VEL
LIN {X 0,Y 418.283,Z 632.549,A -85,B 0,C 180,E1 -10129.428,E2 -10129.428} C_VEL
LIN {X 0,Y 419.036,Z 637,A -85,B 0,C 180,E1 -10132.025,E2 -10132.025} C_VEL
LIN {X 0,Y 419.457,Z 640.706,A -85,B 0,C 180,E1 -10134.097,E2 -10134.097} C_VEL
LIN {X 0,Y 419.282,Z 645.082,A -85,B 0,C 180,E1 -10136.418,E2 -10136.418} C_VEL
LIN {X 0,Y 418.827,Z 651.646,A -85,B 0,C 180,E1 -10139.775,E2 -10139.775} C_VEL
LIN {X 0,Y 418.421,Z 658.231,A -85,B 0,C 180,E1 -10143.032,E2 -10143.032} C_VEL
LIN {X 0,Y 418.066,Z 664.798,A -85,B 0,C 180,E1 -10146.206,E2 -10146.206} C_VEL
LIN {X 0,Y 417.823,Z 671.383,A -85,B 0,C 180,E1 -10149.316,E2 -10149.316} C_VEL
LIN {X 0,Y 417.581,Z 678.904,A -85,B 0,C 180,E1 -10152.792,E2 -10152.792} C_VEL
LIN {X 0,Y 419.923,Z 692.648,A -85,B 0,C 180,E1 -10153.319,E2 -10153.319} C_VEL
LIN {X 0,Y 421.633,Z 705.216,A -85,B 0,C 180,E1 -10153.978,E2 -10153.978} C_VEL
LIN {X 0,Y 420.951,Z 717.736,A -85,B 0,C 180,E1 -10154.755,E2 -10154.755} C_VEL
LIN {X 0,Y 420.228,Z 729.236,A -85,B 0,C 180,E1 -10155.689,E2 -10155.689} C_VEL
LIN {X 0,Y 419.52,Z 740.147,A -85,B 0,C 180,E1 -10156.806,E2 -10156.806} C_VEL
LIN {X 0,Y 418.916,Z 748.818,A -85,B 0,C 180,E1 -10157.895,E2 -10157.895} C_VEL
LIN {X 0,Y 418.332,Z 756.813,A -85,B 0,C 180,E1 -10159.106,E2 -10159.106} C_VEL
LIN {X 0,Y 417.811,Z 764.645,A -85,B 0,C 180,E1 -10160.561,E2 -10160.561} C_VEL
LIN {X 0,Y 417.499,Z 769.979,A -85,B 0,C 180,E1 -10161.774,E2 -10161.774} C_VEL
LIN {X 0,Y 417.236,Z 775.167,A -85,B 0,C 180,E1 -10163.229,E2 -10163.229} C_VEL
LIN {X 0,Y 417.144,Z 779.19,A -85,B 0,C 180,E1 -10164.684,E2 -10164.684} C_VEL
LIN {X 0,Y 417.02,Z 782.155,A -85,B 0,C 180,E1 -10166.135,E2 -10166.135} C_VEL
LIN {X 0,Y 417.023,Z 783.577,A -85,B 0,C 180,E1 -10167.102,E2 -10167.102} C_VEL
LIN {X 0,Y 417.052,Z 784.585,A -85,B 0,C 180,E1 -10168.069,E2 -10168.069} C_VEL
LIN {X 0,Y 417.004,Z 785.42,A -85,B 0,C 180,E1 -10170,E2 -10170} C_VEL
LIN {X 0,Y 417.01,Z 785.206,A -85,B 0,C 180,E1 -10170.966,E2 -10170.966} C_VEL
LIN {X 0,Y 417.052,Z 784.592,A -85,B 0,C 180,E1 -10171.932,E2 -10171.932} C_VEL
LIN {X 0,Y 417.022,Z 783.583,A -85,B 0,C 180,E1 -10172.898,E2 -10172.898} C_VEL
LIN {X 0,Y 417.021,Z 782.172,A -85,B 0,C 180,E1 -10173.866,E2 -10173.866} C_VEL
LIN {X 0,Y 417.147,Z 779.208,A -85,B 0,C 180,E1 -10175.317,E2 -10175.317} C_VEL
LIN {X 0,Y 417.266,Z 775.198,A -85,B 0,C 180,E1 -10176.771,E2 -10176.771} C_VEL
LIN {X 0,Y 417.549,Z 769.038,A -85,B 0,C 180,E1 -10178.469,E2 -10178.469} C_VEL
LIN {X 0,Y 417.964,Z 762.311,A -85,B 0,C 180,E1 -10179.925,E2 -10179.925} C_VEL
LIN {X 0,Y 418.527,Z 753.988,A -85,B 0,C 180,E1 -10181.38,E2 -10181.38} C_VEL
LIN {X 0,Y 419.253,Z 745.473,A -85,B 0,C 180,E1 -10182.587,E2 -10182.587} C_VEL
LIN {X 0,Y 419.892,Z 734.947,A -85,B 0,C 180,E1 -10183.802,E2 -10183.802} C_VEL
LIN {X 0,Y 420.661,Z 723.21,A -85,B 0,C 180,E1 -10184.885,E2 -10184.885} C_VEL
LIN {X 0,Y 421.428,Z 711.454,A -85,B 0,C 180,E1 -10185.724,E2 -10185.724} C_VEL
LIN {X 0,Y 421.606,Z 704.182,A -85,B 0,C 180,E1 -10186.152,E2 -10186.152} C_VEL
LIN {X 0,Y 419.836,Z 691.005,A -85,B 0,C 180,E1 -10186.841,E2 -10186.841} C_VEL
LIN {X 0,Y 417.545,Z 678.29,A -85,B 0,C 180,E1 -10187.352,E2 -10187.352} C_VEL
LIN {X 0,Y 417.815,Z 671.086,A -85,B 0,C 180,E1 -10190.686,E2 -10190.686} C_VEL
LIN {X 0,Y 418.032,Z 664.538,A -85,B 0,C 180,E1 -10193.797,E2 -10193.797} C_VEL
LIN {X 0,Y 418.442,Z 657.764,A -85,B 0,C 180,E1 -10197.105,E2 -10197.105} C_VEL
LIN {X 0,Y 418.801,Z 651.619,A -85,B 0,C 180,E1 -10200.228,E2 -10200.228} C_VEL
LIN {X 0,Y 419.306,Z 645.331,A -85,B 0,C 180,E1 -10203.581,E2 -10203.581} C_VEL
LIN {X 0,Y 419.469,Z 641.221,A -85,B 0,C 180,E1 -10205.903,E2 -10205.903} C_VEL
LIN {X 0,Y 419.061,Z 637.182,A -85,B 0,C 180,E1 -10208.354,E2 -10208.354} C_VEL
LIN {X 0,Y 418.262,Z 632.389,A -85,B 0,C 180,E1 -10211.584,E2 -10211.584} C_VEL
LIN {X 0,Y 418.24,Z 632.39,A -85,B 0,C 180,E1 -10215.109,E2 -10215.109} C_VEL
LIN {X 0,Y 418.242,Z 632.39,A -85,B 0,C 180,E1 -10217.767,E2 -10217.767} C_VEL
LIN {X 0,Y 418.256,Z 632.39,A -85,B 0,C 180,E1 -10220.619,E2 -10220.619} C_VEL
LIN {X 0,Y 418.245,Z 632.389,A -85,B 0,C 180,E1 -10223.976,E2 -10223.976} C_VEL
LIN {X 0,Y 418.259,Z 632.388,A -85,B 0,C 180,E1 -10227.156,E2 -10227.156} C_VEL
LIN {X 0,Y 418.27,Z 632.385,A -85,B 0,C 180,E1 -10230.895,E2 -10230.895} C_VEL
LIN {X 0,Y 418.272,Z 632.383,A -85,B 0,C 180,E1 -10234.096,E2 -10234.096} C_VEL
LIN {X 0,Y 418.24,Z 632.39,A -85,B 0,C 180,E1 -10237.264,E2 -10237.264} C_VEL
LIN {X 0,Y 418.285,Z 632.383,A -85,B 0,C 180,E1 -10240.364,E2 -10240.364} C_VEL
LIN {X 0,Y 418.319,Z 632.38,A -85,B 0,C 180,E1 -10243.405,E2 -10243.405} C_VEL
LIN {X 0,Y 418.348,Z 632.376,A -85,B 0,C 180,E1 -10246.999,E2 -10246.999} C_VEL
LIN {X 0,Y 418.343,Z 632.374,A -85,B 0,C 180,E1 -10250.329,E2 -10250.329} C_VEL
LIN {X 0,Y 418.515,Z 632.353,A -85,B 0,C 180,E1 -10252.279,E2 -10252.279} C_VEL
LIN {X 0,Y 418.515,Z 632.353,A -85,B 0,C 180,E1 -10254.217,E2 -10254.217} C_VEL
LIN {X 0,Y 418.544,Z 632.352,A -85,B 0,C 180,E1 -10258.075,E2 -10258.075} C_VEL
LIN {X 0,Y 418.674,Z 632.335,A -85,B 0,C 180,E1 -10260,E2 -10260} C_VEL
LIN {X 0,Y 418.513,Z 632.357,A -85,B 0,C 180,E1 -10262.888,E2 -10262.888} C_VEL
LIN {X 0,Y 418.494,Z 632.359,A -85,B 0,C 180,E1 -10266.751,E2 -10266.751} C_VEL
LIN {X 0,Y 418.468,Z 632.362,A -85,B 0,C 180,E1 -10267.744,E2 -10267.744} C_VEL
LIN {X 0,Y 418.409,Z 632.749,A -85,B 0,C 180,E1 -10268.695,E2 -10268.695} C_VEL
LIN {X 0,Y 418.271,Z 636.154,A -85,B 0,C 180,E1 -10271.632,E2 -10271.632} C_VEL
LIN {X 0,Y 418.085,Z 639.763,A -85,B 0,C 180,E1 -10274.605,E2 -10274.605} C_VEL
LIN {X 0,Y 417.864,Z 643.558,A -85,B 0,C 180,E1 -10277.622,E2 -10277.622} C_VEL
LIN {X 0,Y 417.683,Z 647.51,A -85,B 0,C 180,E1 -10280.692,E2 -10280.692} C_VEL
LIN {X 0,Y 417.508,Z 651.644,A -85,B 0,C 180,E1 -10283.828,E2 -10283.828} C_VEL
LIN {X 0,Y 417.39,Z 655.986,A -85,B 0,C 180,E1 -10287.041,E2 -10287.041} C_VEL
LIN {X 0,Y 417.343,Z 656.914,A -85,B 0,C 180,E1 -10287.723,E2 -10287.723} C_VEL
LIN {X 0,Y 420.766,Z 671.702,A -85,B 0,C 180,E1 -10288.413,E2 -10288.413} C_VEL
LIN {X 0,Y 422.191,Z 679.701,A -85,B 0,C 180,E1 -10288.865,E2 -10288.865} C_VEL
LIN {X 0,Y 421.564,Z 691.668,A -85,B 0,C 180,E1 -10289.59,E2 -10289.59} C_VEL
LIN {X 0,Y 420.881,Z 703.026,A -85,B 0,C 180,E1 -10290.478,E2 -10290.478} C_VEL
LIN {X 0,Y 420.173,Z 713.021,A -85,B 0,C 180,E1 -10291.455,E2 -10291.455} C_VEL
LIN {X 0,Y 419.458,Z 722.324,A -85,B 0,C 180,E1 -10292.573,E2 -10292.573} C_VEL
LIN {X 0,Y 418.849,Z 731.08,A -85,B 0,C 180,E1 -10293.865,E2 -10293.865} C_VEL
LIN {X 0,Y 418.299,Z 738.14,A -85,B 0,C 180,E1 -10295.131,E2 -10295.131} C_VEL
LIN {X 0,Y 417.782,Z 745.205,A -85,B 0,C 180,E1 -10296.697,E2 -10296.697} C_VEL
LIN {X 0,Y 417.472,Z 750.167,A -85,B 0,C 180,E1 -10298.088,E2 -10298.088} C_VEL
LIN {X 0,Y 417.246,Z 754.826,A -85,B 0,C 180,E1 -10299.797,E2 -10299.797} C_VEL
LIN {X 0,Y 417.095,Z 757.397,A -85,B 0,C 180,E1 -10301.083,E2 -10301.083} C_VEL
LIN {X 0,Y 416.941,Z 759.218,A -85,B 0,C 180,E1 -10302.396,E2 -10302.396} C_VEL
LIN {X 0,Y 416.903,Z 760.311,A -85,B 0,C 180,E1 -10303.722,E2 -10303.722} C_VEL
LIN {X 0,Y 416.891,Z 760.668,A -85,B 0,C 180,E1 -10305.076,E2 -10305.076} C_VEL
LIN {X 0,Y 416.865,Z 760.198,A -85,B 0,C 180,E1 -10306.465,E2 -10306.465} C_VEL
LIN {X 0,Y 416.939,Z 758.868,A -85,B 0,C 180,E1 -10307.874,E2 -10307.874} C_VEL
LIN {X 0,Y 417.129,Z 756.631,A -85,B 0,C 180,E1 -10309.305,E2 -10309.305} C_VEL
LIN {X 0,Y 417.298,Z 753.332,A -85,B 0,C 180,E1 -10310.78,E2 -10310.78} C_VEL
LIN {X 0,Y 417.543,Z 748.822,A -85,B 0,C 180,E1 -10312.288,E2 -10312.288} C_VEL
LIN {X 0,Y 417.905,Z 742.409,A -85,B 0,C 180,E1 -10313.942,E2 -10313.942} C_VEL
LIN {X 0,Y 418.401,Z 735.216,A -85,B 0,C 180,E1 -10315.393,E2 -10315.393} C_VEL
LIN {X 0,Y 419.019,Z 727.148,A -85,B 0,C 180,E1 -10316.714,E2 -10316.714} C_VEL
LIN {X 0,Y 419.675,Z 717.661,A -85,B 0,C 180,E1 -10317.983,E2 -10317.983} C_VEL
LIN {X 0,Y 420.398,Z 707.635,A -85,B 0,C 180,E1 -10319.065,E2 -10319.065} C_VEL
LIN {X 0,Y 421.039,Z 696.53,A -85,B 0,C 180,E1 -10320.028,E2 -10320.028} C_VEL
LIN {X 0,Y 421.728,Z 684.756,A -85,B 0,C 180,E1 -10320.827,E2 -10320.827} C_VEL
LIN {X 0,Y 421.931,Z 678.917,A -85,B 0,C 180,E1 -10321.153,E2 -10321.153} C_VEL
LIN {X 0,Y 419.679,Z 667.205,A -85,B 0,C 180,E1 -10321.775,E2 -10321.775} C_VEL
LIN {X 0,Y 417.28,Z 656.294,A -85,B 0,C 180,E1 -10322.238,E2 -10322.238} C_VEL
LIN {X 0,Y 417.368,Z 651.853,A -85,B 0,C 180,E1 -10325.409,E2 -10325.409} C_VEL
LIN {X 0,Y 417.538,Z 647.908,A -85,B 0,C 180,E1 -10328.265,E2 -10328.265} C_VEL
LIN {X 0,Y 417.675,Z 643.721,A -85,B 0,C 180,E1 -10331.355,E2 -10331.355} C_VEL
LIN {X 0,Y 417.876,Z 639.676,A -85,B 0,C 180,E1 -10334.389,E2 -10334.389} C_VEL
LIN {X 0,Y 418.101,Z 635.781,A -85,B 0,C 180,E1 -10337.377,E2 -10337.377} C_VEL
LIN {X 0,Y 418.141,Z 633.275,A -85,B 0,C 180,E1 -10339.345,E2 -10339.345} C_VEL
LIN {X 0,Y 418.203,Z 632.393,A -85,B 0,C 180,E1 -10340.325,E2 -10340.325} C_VEL
LIN {X 0,Y 418.494,Z 632.357,A -85,B 0,C 180,E1 -10343.249,E2 -10343.249} C_VEL
LIN {X 0,Y 418.342,Z 632.376,A -85,B 0,C 180,E1 -10345.181,E2 -10345.181} C_VEL
LIN {X 0,Y 418.512,Z 632.352,A -85,B 0,C 180,E1 -10347.464,E2 -10347.464} C_VEL
LIN {X 0,Y 417.853,Z 632.435,A -85,B 0,C 180,E1 -10348.268,E2 -10348.268} C_VEL
LIN {X 0,Y 414.975,Z 632.793,A -85,B 0,C 180,E1 -10349.575,E2 -10349.575} C_VEL
LIN {X 0,Y 412.557,Z 633.097,A -85,B 0,C 180,E1 -10350.631,E2 -10350.631} C_VEL
LIN {X 0,Y 411.555,Z 633.22,A -85,B 0,C 180,E1 -10351.447,E2 -10351.447} C_VEL
LIN {X 0,Y 411.494,Z 633.226,A -85,B 0,C 180,E1 -10351.723,E2 -10351.723} C_VEL
LIN {X 0,Y 411.312,Z 633.253,A -85,B 0,C 180,E1 -10354.901,E2 -10354.901} C_VEL
LIN {X 0,Y 411.425,Z 633.239,A -85,B 0,C 180,E1 -10356.867,E2 -10356.867} C_VEL
LIN {X 0,Y 411.093,Z 633.276,A -85,B 0,C 180,E1 -10359.843,E2 -10359.843} C_VEL
LIN {X 0,Y 410.729,Z 633.526,A -85,B 0,C 180,E1 -10362.056,E2 -10362.056} C_VEL
LIN {X 0,Y 410.515,Z 639.446,A -85,B 0,C 180,E1 -10365.897,E2 -10365.897} C_VEL
LIN {X 0,Y 410.357,Z 645.198,A -85,B 0,C 180,E1 -10369.616,E2 -10369.616} C_VEL
LIN {X 0,Y 410.21,Z 650.713,A -85,B 0,C 180,E1 -10373.206,E2 -10373.206} C_VEL
LIN {X 0,Y 410.128,Z 655.946,A -85,B 0,C 180,E1 -10376.598,E2 -10376.598} C_VEL
LIN {X 0,Y 413.094,Z 669.581,A -85,B 0,C 180,E1 -10377.183,E2 -10377.183} C_VEL
LIN {X 0,Y 415.052,Z 680.465,A -85,B 0,C 180,E1 -10377.789,E2 -10377.789} C_VEL
LIN {X 0,Y 414.386,Z 692.692,A -85,B 0,C 180,E1 -10378.558,E2 -10378.558} C_VEL
LIN {X 0,Y 413.626,Z 704.505,A -85,B 0,C 180,E1 -10379.52,E2 -10379.52} C_VEL
LIN {X 0,Y 412.885,Z 714.844,A -85,B 0,C 180,E1 -10380.585,E2 -10380.585} C_VEL
LIN {X 0,Y 412.109,Z 725.195,A -85,B 0,C 180,E1 -10381.915,E2 -10381.915} C_VEL
LIN {X 0,Y 411.491,Z 733.254,A -85,B 0,C 180,E1 -10383.187,E2 -10383.187} C_VEL
LIN {X 0,Y 411.01,Z 740.449,A -85,B 0,C 180,E1 -10384.58,E2 -10384.58} C_VEL
LIN {X 0,Y 410.626,Z 746.358,A -85,B 0,C 180,E1 -10385.995,E2 -10385.995} C_VEL
LIN {X 0,Y 410.294,Z 751.093,A -85,B 0,C 180,E1 -10387.406,E2 -10387.406} C_VEL
LIN {X 0,Y 410.099,Z 754.575,A -85,B 0,C 180,E1 -10388.719,E2 -10388.719} C_VEL
LIN {X 0,Y 409.959,Z 756.276,A -85,B 0,C 180,E1 -10389.516,E2 -10389.516} C_VEL
LIN {X 0,Y 409.795,Z 758.695,A -85,B 0,C 180,E1 -10391.009,E2 -10391.009} C_VEL
LIN {X 0,Y 409.766,Z 760.139,A -85,B 0,C 180,E1 -10392.48,E2 -10392.48} C_VEL
LIN {X 0,Y 409.761,Z 760.669,A -85,B 0,C 180,E1 -10393.915,E2 -10393.915} C_VEL
LIN {X 0,Y 409.795,Z 760.366,A -85,B 0,C 180,E1 -10395.319,E2 -10395.319} C_VEL
LIN {X 0,Y 409.846,Z 759.293,A -85,B 0,C 180,E1 -10396.692,E2 -10396.692} C_VEL
LIN {X 0,Y 409.938,Z 757.48,A -85,B 0,C 180,E1 -10398.039,E2 -10398.039} C_VEL
LIN {X 0,Y 410.205,Z 753.523,A -85,B 0,C 180,E1 -10399.937,E2 -10399.937} C_VEL
LIN {X 0,Y 410.54,Z 748.5,A -85,B 0,C 180,E1 -10401.643,E2 -10401.643} C_VEL
LIN {X 0,Y 410.923,Z 742.339,A -85,B 0,C 180,E1 -10403.23,E2 -10403.23} C_VEL
LIN {X 0,Y 411.523,Z 734.611,A -85,B 0,C 180,E1 -10404.805,E2 -10404.805} C_VEL
LIN {X 0,Y 412.256,Z 725.912,A -85,B 0,C 180,E1 -10406.218,E2 -10406.218} C_VEL
LIN {X 0,Y 413.078,Z 715.331,A -85,B 0,C 180,E1 -10407.593,E2 -10407.593} C_VEL
LIN {X 0,Y 413.825,Z 705.08,A -85,B 0,C 180,E1 -10408.66,E2 -10408.66} C_VEL
LIN {X 0,Y 414.638,Z 692.703,A -85,B 0,C 180,E1 -10409.674,E2 -10409.674} C_VEL
LIN {X 0,Y 415.311,Z 680.541,A -85,B 0,C 180,E1 -10410.436,E2 -10410.436} C_VEL
LIN {X 0,Y 412.894,Z 667.656,A -85,B 0,C 180,E1 -10411.157,E2 -10411.157} C_VEL
LIN {X 0,Y 410.214,Z 656.364,A -85,B 0,C 180,E1 -10411.682,E2 -10411.682} C_VEL
LIN {X 0,Y 410.323,Z 650.867,A -85,B 0,C 180,E1 -10415.199,E2 -10415.199} C_VEL
LIN {X 0,Y 410.418,Z 645.029,A -85,B 0,C 180,E1 -10418.924,E2 -10418.924} C_VEL
LIN {X 0,Y 410.502,Z 640.037,A -85,B 0,C 180,E1 -10422.051,E2 -10422.051} C_VEL
LIN {X 0,Y 410.648,Z 635.036,A -85,B 0,C 180,E1 -10425.125,E2 -10425.125} C_VEL
LIN {X 0,Y 410.763,Z 633.326,A -85,B 0,C 180,E1 -10426.267,E2 -10426.267} C_VEL
LIN {X 0,Y 411.171,Z 633.271,A -85,B 0,C 180,E1 -10429.163,E2 -10429.163} C_VEL
LIN {X 0,Y 411.419,Z 633.242,A -85,B 0,C 180,E1 -10432.206,E2 -10432.206} C_VEL
LIN {X 0,Y 411.471,Z 633.234,A -85,B 0,C 180,E1 -10434.118,E2 -10434.118} C_VEL
LIN {X 0,Y 411.511,Z 633.228,A -85,B 0,C 180,E1 -10438.043,E2 -10438.043} C_VEL
LIN {X 0,Y 411.64,Z 633.212,A -85,B 0,C 180,E1 -10440,E2 -10440} C_VEL
LIN {X 0,Y 411.463,Z 633.234,A -85,B 0,C 180,E1 -10442.937,E2 -10442.937} C_VEL
LIN {X 0,Y 411.457,Z 633.234,A -85,B 0,C 180,E1 -10446.867,E2 -10446.867} C_VEL
LIN {X 0,Y 411.291,Z 633.254,A -85,B 0,C 180,E1 -10449.839,E2 -10449.839} C_VEL
LIN {X 0,Y 411.301,Z 633.253,A -85,B 0,C 180,E1 -10453.104,E2 -10453.104} C_VEL
LIN {X 0,Y 411.253,Z 633.259,A -85,B 0,C 180,E1 -10456.889,E2 -10456.889} C_VEL
LIN {X 0,Y 411.227,Z 633.264,A -85,B 0,C 180,E1 -10459.987,E2 -10459.987} C_VEL
LIN {X 0,Y 411.2,Z 633.265,A -85,B 0,C 180,E1 -10463.148,E2 -10463.148} C_VEL
LIN {X 0,Y 411.235,Z 633.26,A -85,B 0,C 180,E1 -10466.381,E2 -10466.381} C_VEL
LIN {X 0,Y 411.208,Z 633.265,A -85,B 0,C 180,E1 -10469.712,E2 -10469.712} C_VEL
LIN {X 0,Y 411.203,Z 633.265,A -85,B 0,C 180,E1 -10473.156,E2 -10473.156} C_VEL
LIN {X 0,Y 411.192,Z 633.267,A -85,B 0,C 180,E1 -10476.554,E2 -10476.554} C_VEL
LIN {X 0,Y 411.213,Z 633.262,A -85,B 0,C 180,E1 -10479.729,E2 -10479.729} C_VEL
LIN {X 0,Y 411.171,Z 633.27,A -85,B 0,C 180,E1 -10483.134,E2 -10483.134} C_VEL
LIN {X 0,Y 411.166,Z 633.271,A -85,B 0,C 180,E1 -10485.882,E2 -10485.882} C_VEL
LIN {X 0,Y 411.228,Z 633.314,A -85,B 0,C 180,E1 -10489.138,E2 -10489.138} C_VEL
LIN {X 0,Y 412.073,Z 638.341,A -85,B 0,C 180,E1 -10492.122,E2 -10492.122} C_VEL
LIN {X 0,Y 412.459,Z 642.721,A -85,B 0,C 180,E1 -10494.597,E2 -10494.597} C_VEL
LIN {X 0,Y 412.08,Z 648.201,A -85,B 0,C 180,E1 -10497.505,E2 -10497.505} C_VEL
LIN {X 0,Y 411.725,Z 654.033,A -85,B 0,C 180,E1 -10500.523,E2 -10500.523} C_VEL
LIN {X 0,Y 411.226,Z 661.318,A -85,B 0,C 180,E1 -10504.164,E2 -10504.164} C_VEL
LIN {X 0,Y 410.92,Z 668.071,A -85,B 0,C 180,E1 -10507.454,E2 -10507.454} C_VEL
LIN {X 0,Y 410.626,Z 673.987,A -85,B 0,C 180,E1 -10510.279,E2 -10510.279} C_VEL
LIN {X 0,Y 410.506,Z 678.712,A -85,B 0,C 180,E1 -10512.504,E2 -10512.504} C_VEL
LIN {X 0,Y 412.953,Z 692.91,A -85,B 0,C 180,E1 -10513.068,E2 -10513.068} C_VEL
LIN {X 0,Y 414.733,Z 706.499,A -85,B 0,C 180,E1 -10513.804,E2 -10513.804} C_VEL
LIN {X 0,Y 413.966,Z 718.971,A -85,B 0,C 180,E1 -10514.618,E2 -10514.618} C_VEL
LIN {X 0,Y 413.229,Z 730.377,A -85,B 0,C 180,E1 -10515.587,E2 -10515.587} C_VEL
LIN {X 0,Y 412.49,Z 740.889,A -85,B 0,C 180,E1 -10516.703,E2 -10516.703} C_VEL
LIN {X 0,Y 411.808,Z 750.258,A -85,B 0,C 180,E1 -10517.933,E2 -10517.933} C_VEL
LIN {X 0,Y 411.113,Z 759.319,A -85,B 0,C 180,E1 -10519.411,E2 -10519.411} C_VEL
LIN {X 0,Y 410.653,Z 766.627,A -85,B 0,C 180,E1 -10520.892,E2 -10520.892} C_VEL
LIN {X 0,Y 410.336,Z 771.568,A -85,B 0,C 180,E1 -10522.125,E2 -10522.125} C_VEL
LIN {X 0,Y 410.054,Z 776.819,A -85,B 0,C 180,E1 -10523.761,E2 -10523.761} C_VEL
LIN {X 0,Y 410.034,Z 780.035,A -85,B 0,C 180,E1 -10525.084,E2 -10525.084} C_VEL
LIN {X 0,Y 409.939,Z 781.926,A -85,B 0,C 180,E1 -10526.068,E2 -10526.068} C_VEL
LIN {X 0,Y 409.921,Z 783.355,A -85,B 0,C 180,E1 -10527.052,E2 -10527.052} C_VEL
LIN {X 0,Y 409.963,Z 784.366,A -85,B 0,C 180,E1 -10528.036,E2 -10528.036} C_VEL
LIN {X 0,Y 409.935,Z 784.983,A -85,B 0,C 180,E1 -10529.018,E2 -10529.018} C_VEL
LIN {X 0,Y 409.926,Z 785.208,A -85,B 0,C 180,E1 -10530,E2 -10530} C_VEL
LIN {X 0,Y 409.935,Z 784.999,A -85,B 0,C 180,E1 -10530.983,E2 -10530.983} C_VEL
LIN {X 0,Y 409.963,Z 784.386,A -85,B 0,C 180,E1 -10531.965,E2 -10531.965} C_VEL
LIN {X 0,Y 409.939,Z 781.97,A -85,B 0,C 180,E1 -10533.933,E2 -10533.933} C_VEL
LIN {X 0,Y 410.044,Z 779.01,A -85,B 0,C 180,E1 -10535.41,E2 -10535.41} C_VEL
LIN {X 0,Y 410.191,Z 775.008,A -85,B 0,C 180,E1 -10536.889,E2 -10536.889} C_VEL
LIN {X 0,Y 410.498,Z 768.864,A -85,B 0,C 180,E1 -10538.616,E2 -10538.616} C_VEL
LIN {X 0,Y 410.948,Z 762.154,A -85,B 0,C 180,E1 -10540.096,E2 -10540.096} C_VEL
LIN {X 0,Y 411.552,Z 753.841,A -85,B 0,C 180,E1 -10541.575,E2 -10541.575} C_VEL
LIN {X 0,Y 412.307,Z 745.344,A -85,B 0,C 180,E1 -10542.803,E2 -10542.803} C_VEL
LIN {X 0,Y 412.98,Z 734.576,A -85,B 0,C 180,E1 -10544.066,E2 -10544.066} C_VEL
LIN {X 0,Y 413.787,Z 723.131,A -85,B 0,C 180,E1 -10545.138,E2 -10545.138} C_VEL
LIN {X 0,Y 414.605,Z 711.502,A -85,B 0,C 180,E1 -10545.985,E2 -10545.985} C_VEL
LIN {X 0,Y 414.794,Z 705.494,A -85,B 0,C 180,E1 -10546.351,E2 -10546.351} C_VEL
LIN {X 0,Y 413.013,Z 691.94,A -85,B 0,C 180,E1 -10547.096,E2 -10547.096} C_VEL
LIN {X 0,Y 410.607,Z 679.1,A -85,B 0,C 180,E1 -10547.632,E2 -10547.632} C_VEL
LIN {X 0,Y 410.469,Z 678.031,A -85,B 0,C 180,E1 -10547.693,E2 -10547.693} C_VEL
LIN {X 0,Y 410.774,Z 670.925,A -85,B 0,C 180,E1 -10551.057,E2 -10551.057} C_VEL
LIN {X 0,Y 411.035,Z 664.405,A -85,B 0,C 180,E1 -10554.228,E2 -10554.228} C_VEL
LIN {X 0,Y 411.429,Z 657.955,A -85,B 0,C 180,E1 -10557.466,E2 -10557.466} C_VEL
LIN {X 0,Y 411.823,Z 651.582,A -85,B 0,C 180,E1 -10560.795,E2 -10560.795} C_VEL
LIN {X 0,Y 412.403,Z 645.328,A -85,B 0,C 180,E1 -10564.22,E2 -10564.22} C_VEL
LIN {X 0,Y 412.391,Z 640.983,A -85,B 0,C 180,E1 -10566.776,E2 -10566.776} C_VEL
LIN {X 0,Y 411.727,Z 636.248,A -85,B 0,C 180,E1 -10569.813,E2 -10569.813} C_VEL
LIN {X 0,Y 411.216,Z 633.267,A -85,B 0,C 180,E1 -10571.965,E2 -10571.965} C_VEL
LIN {X 0,Y 411.179,Z 633.269,A -85,B 0,C 180,E1 -10575.51,E2 -10575.51} C_VEL
LIN {X 0,Y 411.166,Z 633.272,A -85,B 0,C 180,E1 -10578.772,E2 -10578.772} C_VEL
LIN {X 0,Y 411.206,Z 633.266,A -85,B 0,C 180,E1 -10581.831,E2 -10581.831} C_VEL
LIN {X 0,Y 411.213,Z 633.265,A -85,B 0,C 180,E1 -10585.121,E2 -10585.121} C_VEL
LIN {X 0,Y 411.167,Z 633.269,A -85,B 0,C 180,E1 -10588.003,E2 -10588.003} C_VEL
LIN {X 0,Y 411.22,Z 633.262,A -85,B 0,C 180,E1 -10591.41,E2 -10591.41} C_VEL
LIN {X 0,Y 411.24,Z 633.259,A -85,B 0,C 180,E1 -10593.619,E2 -10593.619} C_VEL
LIN {X 0,Y 411.205,Z 633.266,A -85,B 0,C 180,E1 -10596.853,E2 -10596.853} C_VEL
LIN {X 0,Y 411.217,Z 633.263,A -85,B 0,C 180,E1 -10600.05,E2 -10600.05} C_VEL
LIN {X 0,Y 411.265,Z 633.258,A -85,B 0,C 180,E1 -10603.131,E2 -10603.131} C_VEL
LIN {X 0,Y 411.307,Z 633.253,A -85,B 0,C 180,E1 -10606.896,E2 -10606.896} C_VEL
LIN {X 0,Y 411.295,Z 633.252,A -85,B 0,C 180,E1 -10610.161,E2 -10610.161} C_VEL
LIN {X 0,Y 411.484,Z 633.228,A -85,B 0,C 180,E1 -10612.147,E2 -10612.147} C_VEL
LIN {X 0,Y 411.477,Z 633.23,A -85,B 0,C 180,E1 -10614.118,E2 -10614.118} C_VEL
LIN {X 0,Y 411.513,Z 633.228,A -85,B 0,C 180,E1 -10618.043,E2 -10618.043} C_VEL
LIN {X 0,Y 411.644,Z 633.211,A -85,B 0,C 180,E1 -10620,E2 -10620} C_VEL
LIN {X 0,Y 411.468,Z 633.234,A -85,B 0,C 180,E1 -10622.937,E2 -10622.937} C_VEL
LIN {X 0,Y 411.458,Z 633.235,A -85,B 0,C 180,E1 -10626.867,E2 -10626.867} C_VEL
LIN {X 0,Y 411.415,Z 633.241,A -85,B 0,C 180,E1 -10627.855,E2 -10627.855} C_VEL
LIN {X 0,Y 411.381,Z 635.114,A -85,B 0,C 180,E1 -10629.837,E2 -10629.837} C_VEL
LIN {X 0,Y 411.157,Z 638.795,A -85,B 0,C 180,E1 -10633.014,E2 -10633.014} C_VEL
LIN {X 0,Y 410.949,Z 642.282,A -85,B 0,C 180,E1 -10635.88,E2 -10635.88} C_VEL
LIN {X 0,Y 410.734,Z 647.141,A -85,B 0,C 180,E1 -10639.763,E2 -10639.763} C_VEL
LIN {X 0,Y 410.487,Z 651.563,A -85,B 0,C 180,E1 -10643.19,E2 -10643.19} C_VEL
LIN {X 0,Y 410.345,Z 655.874,A -85,B 0,C 180,E1 -10646.443,E2 -10646.443} C_VEL
LIN {X 0,Y 410.315,Z 657.16,A -85,B 0,C 180,E1 -10647.399,E2 -10647.399} C_VEL
LIN {X 0,Y 413.715,Z 671.637,A -85,B 0,C 180,E1 -10648.091,E2 -10648.091} C_VEL
LIN {X 0,Y 415.371,Z 680.704,A -85,B 0,C 180,E1 -10648.623,E2 -10648.623} C_VEL
LIN {X 0,Y 414.622,Z 693.715,A -85,B 0,C 180,E1 -10649.443,E2 -10649.443} C_VEL
LIN {X 0,Y 413.966,Z 704.13,A -85,B 0,C 180,E1 -10650.296,E2 -10650.296} C_VEL
LIN {X 0,Y 413.12,Z 715.416,A -85,B 0,C 180,E1 -10651.461,E2 -10651.461} C_VEL
LIN {X 0,Y 412.329,Z 725.528,A -85,B 0,C 180,E1 -10652.763,E2 -10652.763} C_VEL
LIN {X 0,Y 411.699,Z 733.489,A -85,B 0,C 180,E1 -10654.028,E2 -10654.028} C_VEL
LIN {X 0,Y 411.082,Z 741.185,A -85,B 0,C 180,E1 -10655.541,E2 -10655.541} C_VEL
LIN {X 0,Y 410.618,Z 747.512,A -85,B 0,C 180,E1 -10657.101,E2 -10657.101} C_VEL
LIN {X 0,Y 410.308,Z 752.556,A -85,B 0,C 180,E1 -10658.697,E2 -10658.697} C_VEL
LIN {X 0,Y 410.13,Z 755.827,A -85,B 0,C 180,E1 -10660.06,E2 -10660.06} C_VEL
LIN {X 0,Y 410.007,Z 757.684,A -85,B 0,C 180,E1 -10661.043,E2 -10661.043} C_VEL
LIN {X 0,Y 409.863,Z 759.608,A -85,B 0,C 180,E1 -10662.495,E2 -10662.495} C_VEL
LIN {X 0,Y 409.803,Z 760.633,A -85,B 0,C 180,E1 -10663.922,E2 -10663.922} C_VEL
LIN {X 0,Y 409.787,Z 760.835,A -85,B 0,C 180,E1 -10665.318,E2 -10665.318} C_VEL
LIN {X 0,Y 409.777,Z 760.274,A -85,B 0,C 180,E1 -10666.683,E2 -10666.683} C_VEL
LIN {X 0,Y 409.857,Z 758.941,A -85,B 0,C 180,E1 -10668.029,E2 -10668.029} C_VEL
LIN {X 0,Y 410.039,Z 756.851,A -85,B 0,C 180,E1 -10669.359,E2 -10669.359} C_VEL
LIN {X 0,Y 410.197,Z 754.063,A -85,B 0,C 180,E1 -10670.659,E2 -10670.659} C_VEL
LIN {X 0,Y 410.461,Z 749.392,A -85,B 0,C 180,E1 -10672.289,E2 -10672.289} C_VEL
LIN {X 0,Y 410.844,Z 743.002,A -85,B 0,C 180,E1 -10673.99,E2 -10673.99} C_VEL
LIN {X 0,Y 411.334,Z 736.247,A -85,B 0,C 180,E1 -10675.405,E2 -10675.405} C_VEL
LIN {X 0,Y 412.069,Z 727.185,A -85,B 0,C 180,E1 -10676.922,E2 -10676.922} C_VEL
LIN {X 0,Y 412.684,Z 718.286,A -85,B 0,C 180,E1 -10678.134,E2 -10678.134} C_VEL
LIN {X 0,Y 413.419,Z 708.76,A -85,B 0,C 180,E1 -10679.195,E2 -10679.195} C_VEL
LIN {X 0,Y 414.051,Z 698.692,A -85,B 0,C 180,E1 -10680.11,E2 -10680.11} C_VEL
LIN {X 0,Y 414.806,Z 686.364,A -85,B 0,C 180,E1 -10680.988,E2 -10680.988} C_VEL
LIN {X 0,Y 414.943,Z 679.108,A -85,B 0,C 180,E1 -10681.414,E2 -10681.414} C_VEL
LIN {X 0,Y 412.438,Z 666.46,A -85,B 0,C 180,E1 -10682.091,E2 -10682.091} C_VEL
LIN {X 0,Y 410.204,Z 656.481,A -85,B 0,C 180,E1 -10682.524,E2 -10682.524} C_VEL
LIN {X 0,Y 410.307,Z 652.061,A -85,B 0,C 180,E1 -10685.727,E2 -10685.727} C_VEL
LIN {X 0,Y 410.51,Z 647.705,A -85,B 0,C 180,E1 -10688.929,E2 -10688.929} C_VEL
LIN {X 0,Y 410.677,Z 643.538,A -85,B 0,C 180,E1 -10692.059,E2 -10692.059} C_VEL
LIN {X 0,Y 410.864,Z 639.515,A -85,B 0,C 180,E1 -10695.132,E2 -10695.132} C_VEL
LIN {X 0,Y 411.071,Z 635.646,A -85,B 0,C 180,E1 -10698.161,E2 -10698.161} C_VEL
LIN {X 0,Y 411.126,Z 633.275,A -85,B 0,C 180,E1 -10700.157,E2 -10700.157} C_VEL
LIN {X 0,Y 411.455,Z 633.235,A -85,B 0,C 180,E1 -10703.133,E2 -10703.133} C_VEL
LIN {X 0,Y 411.313,Z 633.252,A -85,B 0,C 180,E1 -10705.099,E2 -10705.099} C_VEL
LIN {X 0,Y 411.517,Z 633.222,A -85,B 0,C 180,E1 -10708.042,E2 -10708.042} C_VEL
LIN {X 0,Y 411.646,Z 633.207,A -85,B 0,C 180,E1 -10710,E2 -10710} C_VEL
LIN {X 0,Y 411.494,Z 633.226,A -85,B 0,C 180,E1 -10711.723,E2 -10711.723} C_VEL
LIN {X 0,Y 410.886,Z 633.305,A -85,B 0,C 180,E1 -10712.538,E2 -10712.538} C_VEL
LIN {X 0,Y 408.061,Z 633.655,A -85,B 0,C 180,E1 -10713.861,E2 -10713.861} C_VEL
LIN {X 0,Y 405.609,Z 633.963,A -85,B 0,C 180,E1 -10714.93,E2 -10714.93} C_VEL
LIN {X 0,Y 404.516,Z 634.096,A -85,B 0,C 180,E1 -10715.757,E2 -10715.757} C_VEL
LIN {X 0,Y 404.408,Z 634.108,A -85,B 0,C 180,E1 -10716.037,E2 -10716.037} C_VEL
LIN {X 0,Y 404.287,Z 634.124,A -85,B 0,C 180,E1 -10717.994,E2 -10717.994} C_VEL
LIN {X 0,Y 403.838,Z 634.184,A -85,B 0,C 180,E1 -10721.036,E2 -10721.036} C_VEL
LIN {X 0,Y 403.676,Z 634.32,A -85,B 0,C 180,E1 -10722.059,E2 -10722.059} C_VEL
LIN {X 0,Y 403.433,Z 640.627,A -85,B 0,C 180,E1 -10726.184,E2 -10726.184} C_VEL
LIN {X 0,Y 403.296,Z 646.123,A -85,B 0,C 180,E1 -10729.775,E2 -10729.775} C_VEL
LIN {X 0,Y 403.12,Z 652.036,A -85,B 0,C 180,E1 -10733.639,E2 -10733.639} C_VEL
LIN {X 0,Y 403.053,Z 656.088,A -85,B 0,C 180,E1 -10736.295,E2 -10736.295} C_VEL
LIN {X 0,Y 406.276,Z 670.745,A -85,B 0,C 180,E1 -10736.955,E2 -10736.955} C_VEL
LIN {X 0,Y 408.182,Z 681.13,A -85,B 0,C 180,E1 -10737.558,E2 -10737.558} C_VEL
LIN {X 0,Y 407.457,Z 694.01,A -85,B 0,C 180,E1 -10738.397,E2 -10738.397} C_VEL
LIN {X 0,Y 406.674,Z 705.475,A -85,B 0,C 180,E1 -10739.364,E2 -10739.364} C_VEL
LIN {X 0,Y 405.811,Z 716.74,A -85,B 0,C 180,E1 -10740.578,E2 -10740.578} C_VEL
LIN {X 0,Y 405.043,Z 726.573,A -85,B 0,C 180,E1 -10741.897,E2 -10741.897} C_VEL
LIN {X 0,Y 404.427,Z 734.605,A -85,B 0,C 180,E1 -10743.231,E2 -10743.231} C_VEL
LIN {X 0,Y 403.857,Z 741.995,A -85,B 0,C 180,E1 -10744.744,E2 -10744.744} C_VEL
LIN {X 0,Y 403.437,Z 748.138,A -85,B 0,C 180,E1 -10746.319,E2 -10746.319} C_VEL
LIN {X 0,Y 403.199,Z 752.082,A -85,B 0,C 180,E1 -10747.594,E2 -10747.594} C_VEL
LIN {X 0,Y 402.981,Z 755.293,A -85,B 0,C 180,E1 -10748.89,E2 -10748.89} C_VEL
LIN {X 0,Y 402.773,Z 757.797,A -85,B 0,C 180,E1 -10750.211,E2 -10750.211} C_VEL
LIN {X 0,Y 402.676,Z 759.534,A -85,B 0,C 180,E1 -10751.545,E2 -10751.545} C_VEL
LIN {X 0,Y 402.657,Z 760.56,A -85,B 0,C 180,E1 -10752.898,E2 -10752.898} C_VEL
LIN {X 0,Y 402.685,Z 760.864,A -85,B 0,C 180,E1 -10754.31,E2 -10754.31} C_VEL
LIN {X 0,Y 402.7,Z 760.381,A -85,B 0,C 180,E1 -10755.726,E2 -10755.726} C_VEL
LIN {X 0,Y 402.776,Z 759.087,A -85,B 0,C 180,E1 -10757.125,E2 -10757.125} C_VEL
LIN {X 0,Y 402.914,Z 756.864,A -85,B 0,C 180,E1 -10758.593,E2 -10758.593} C_VEL
LIN {X 0,Y 403.148,Z 753.643,A -85,B 0,C 180,E1 -10760.088,E2 -10760.088} C_VEL
LIN {X 0,Y 403.455,Z 749.263,A -85,B 0,C 180,E1 -10761.616,E2 -10761.616} C_VEL
LIN {X 0,Y 403.853,Z 743.518,A -85,B 0,C 180,E1 -10763.178,E2 -10763.178} C_VEL
LIN {X 0,Y 404.446,Z 736.125,A -85,B 0,C 180,E1 -10764.756,E2 -10764.756} C_VEL
LIN {X 0,Y 405.238,Z 727.136,A -85,B 0,C 180,E1 -10766.291,E2 -10766.291} C_VEL
LIN {X 0,Y 405.974,Z 717.993,A -85,B 0,C 180,E1 -10767.544,E2 -10767.544} C_VEL
LIN {X 0,Y 406.881,Z 706.692,A -85,B 0,C 180,E1 -10768.789,E2 -10768.789} C_VEL
LIN {X 0,Y 407.59,Z 696.748,A -85,B 0,C 180,E1 -10769.668,E2 -10769.668} C_VEL
LIN {X 0,Y 408.36,Z 684.975,A -85,B 0,C 180,E1 -10770.485,E2 -10770.485} C_VEL
LIN {X 0,Y 408.331,Z 680.34,A -85,B 0,C 180,E1 -10770.766,E2 -10770.766} C_VEL
LIN {X 0,Y 405.871,Z 667.669,A -85,B 0,C 180,E1 -10771.493,E2 -10771.493} C_VEL
LIN {X 0,Y 403.141,Z 656.567,A -85,B 0,C 180,E1 -10772.015,E2 -10772.015} C_VEL
LIN {X 0,Y 403.285,Z 651.521,A -85,B 0,C 180,E1 -10775.276,E2 -10775.276} C_VEL
LIN {X 0,Y 403.33,Z 646.435,A -85,B 0,C 180,E1 -10778.535,E2 -10778.535} C_VEL
LIN {X 0,Y 403.444,Z 641.465,A -85,B 0,C 180,E1 -10781.726,E2 -10781.726} C_VEL
LIN {X 0,Y 403.576,Z 636.365,A -85,B 0,C 180,E1 -10784.858,E2 -10784.858} C_VEL
LIN {X 0,Y 403.738,Z 634.202,A -85,B 0,C 180,E1 -10786.28,E2 -10786.28} C_VEL
LIN {X 0,Y 404.097,Z 634.152,A -85,B 0,C 180,E1 -10788.971,E2 -10788.971} C_VEL
LIN {X 0,Y 404.397,Z 634.116,A -85,B 0,C 180,E1 -10792.132,E2 -10792.132} C_VEL
LIN {X 0,Y 404.419,Z 634.113,A -85,B 0,C 180,E1 -10794.015,E2 -10794.015} C_VEL
LIN {X 0,Y 404.479,Z 634.104,A -85,B 0,C 180,E1 -10798.008,E2 -10798.008} C_VEL
LIN {X 0,Y 404.61,Z 634.088,A -85,B 0,C 180,E1 -10800,E2 -10800} C_VEL
LIN {X 0,Y 404.42,Z 634.111,A -85,B 0,C 180,E1 -10802.988,E2 -10802.988} C_VEL
LIN {X 0,Y 404.408,Z 634.112,A -85,B 0,C 180,E1 -10806.987,E2 -10806.987} C_VEL
LIN {X 0,Y 404.256,Z 634.13,A -85,B 0,C 180,E1 -10810.012,E2 -10810.012} C_VEL
LIN {X 0,Y 404.262,Z 634.13,A -85,B 0,C 180,E1 -10813.212,E2 -10813.212} C_VEL
LIN {X 0,Y 404.212,Z 634.137,A -85,B 0,C 180,E1 -10817.007,E2 -10817.007} C_VEL
LIN {X 0,Y 404.16,Z 634.143,A -85,B 0,C 180,E1 -10820.352,E2 -10820.352} C_VEL
LIN {X 0,Y 404.166,Z 634.141,A -85,B 0,C 180,E1 -10823.575,E2 -10823.575} C_VEL
LIN {X 0,Y 404.18,Z 634.14,A -85,B 0,C 180,E1 -10825.767,E2 -10825.767} C_VEL
LIN {X 0,Y 404.195,Z 634.139,A -85,B 0,C 180,E1 -10828,E2 -10828} C_VEL
LIN {X 0,Y 404.14,Z 634.145,A -85,B 0,C 180,E1 -10831.559,E2 -10831.559} C_VEL
LIN {X 0,Y 404.182,Z 634.14,A -85,B 0,C 180,E1 -10835.016,E2 -10835.016} C_VEL
LIN {X 0,Y 404.155,Z 634.143,A -85,B 0,C 180,E1 -10838.757,E2 -10838.757} C_VEL
LIN {X 0,Y 404.12,Z 634.147,A -85,B 0,C 180,E1 -10841.6,E2 -10841.6} C_VEL
LIN {X 0,Y 404.143,Z 634.146,A -85,B 0,C 180,E1 -10844.523,E2 -10844.523} C_VEL
LIN {X 0,Y 404.135,Z 634.147,A -85,B 0,C 180,E1 -10847.296,E2 -10847.296} C_VEL
LIN {X 0,Y 404.222,Z 634.284,A -85,B 0,C 180,E1 -10848.973,E2 -10848.973} C_VEL
LIN {X 0,Y 405.034,Z 639.285,A -85,B 0,C 180,E1 -10851.998,E2 -10851.998} C_VEL
LIN {X 0,Y 405.438,Z 643.737,A -85,B 0,C 180,E1 -10854.559,E2 -10854.559} C_VEL
LIN {X 0,Y 405.063,Z 649.101,A -85,B 0,C 180,E1 -10857.463,E2 -10857.463} C_VEL
LIN {X 0,Y 404.607,Z 655.657,A -85,B 0,C 180,E1 -10860.899,E2 -10860.899} C_VEL
LIN {X 0,Y 404.129,Z 663.201,A -85,B 0,C 180,E1 -10864.73,E2 -10864.73} C_VEL
LIN {X 0,Y 403.788,Z 669.876,A -85,B 0,C 180,E1 -10868.025,E2 -10868.025} C_VEL
LIN {X 0,Y 403.475,Z 676.427,A -85,B 0,C 180,E1 -10871.202,E2 -10871.202} C_VEL
LIN {X 0,Y 403.436,Z 678.664,A -85,B 0,C 180,E1 -10872.223,E2 -10872.223} C_VEL
LIN {X 0,Y 405.818,Z 691.93,A -85,B 0,C 180,E1 -10872.749,E2 -10872.749} C_VEL
LIN {X 0,Y 407.519,Z 704.562,A -85,B 0,C 180,E1 -10873.432,E2 -10873.432} C_VEL
LIN {X 0,Y 407.701,Z 710.009,A -85,B 0,C 180,E1 -10873.77,E2 -10873.77} C_VEL
LIN {X 0,Y 406.882,Z 721.649,A -85,B 0,C 180,E1 -10874.6,E2 -10874.6} C_VEL
LIN {X 0,Y 406.093,Z 733.077,A -85,B 0,C 180,E1 -10875.645,E2 -10875.645} C_VEL
LIN {X 0,Y 405.379,Z 742.528,A -85,B 0,C 180,E1 -10876.72,E2 -10876.72} C_VEL
LIN {X 0,Y 404.691,Z 751.549,A -85,B 0,C 180,E1 -10877.972,E2 -10877.972} C_VEL
LIN {X 0,Y 404.002,Z 760.365,A -85,B 0,C 180,E1 -10879.476,E2 -10879.476} C_VEL
LIN {X 0,Y 403.545,Z 767.407,A -85,B 0,C 180,E1 -10880.983,E2 -10880.983} C_VEL
LIN {X 0,Y 403.155,Z 773.035,A -85,B 0,C 180,E1 -10882.488,E2 -10882.488} C_VEL
LIN {X 0,Y 402.967,Z 777.456,A -85,B 0,C 180,E1 -10883.994,E2 -10883.994} C_VEL
LIN {X 0,Y 402.947,Z 779.791,A -85,B 0,C 180,E1 -10884.997,E2 -10884.997} C_VEL
LIN {X 0,Y 402.859,Z 781.69,A -85,B 0,C 180,E1 -10885.999,E2 -10885.999} C_VEL
LIN {X 0,Y 402.821,Z 783.128,A -85,B 0,C 180,E1 -10887,E2 -10887} C_VEL
LIN {X 0,Y 402.861,Z 784.144,A -85,B 0,C 180,E1 -10888.001,E2 -10888.001} C_VEL
LIN {X 0,Y 402.862,Z 784.765,A -85,B 0,C 180,E1 -10889.001,E2 -10889.001} C_VEL
LIN {X 0,Y 402.851,Z 784.996,A -85,B 0,C 180,E1 -10890,E2 -10890} C_VEL
LIN {X 0,Y 402.862,Z 784.795,A -85,B 0,C 180,E1 -10891,E2 -10891} C_VEL
LIN {X 0,Y 402.861,Z 784.184,A -85,B 0,C 180,E1 -10892,E2 -10892} C_VEL
LIN {X 0,Y 402.86,Z 781.779,A -85,B 0,C 180,E1 -10894.002,E2 -10894.002} C_VEL
LIN {X 0,Y 402.946,Z 778.824,A -85,B 0,C 180,E1 -10895.505,E2 -10895.505} C_VEL
LIN {X 0,Y 403.11,Z 774.83,A -85,B 0,C 180,E1 -10897.01,E2 -10897.01} C_VEL
LIN {X 0,Y 403.436,Z 768.699,A -85,B 0,C 180,E1 -10898.768,E2 -10898.768} C_VEL
LIN {X 0,Y 403.938,Z 761.998,A -85,B 0,C 180,E1 -10900.273,E2 -10900.273} C_VEL
LIN {X 0,Y 404.589,Z 753.695,A -85,B 0,C 180,E1 -10901.778,E2 -10901.778} C_VEL
LIN {X 0,Y 405.35,Z 745.214,A -85,B 0,C 180,E1 -10903.026,E2 -10903.026} C_VEL
LIN {X 0,Y 406.02,Z 735.26,A -85,B 0,C 180,E1 -10904.226,E2 -10904.226} C_VEL
LIN {X 0,Y 406.813,Z 724.487,A -85,B 0,C 180,E1 -10905.276,E2 -10905.276} C_VEL
LIN {X 0,Y 407.665,Z 713.422,A -85,B 0,C 180,E1 -10906.133,E2 -10906.133} C_VEL
LIN {X 0,Y 407.891,Z 706.094,A -85,B 0,C 180,E1 -10906.606,E2 -10906.606} C_VEL
LIN {X 0,Y 406.164,Z 692.267,A -85,B 0,C 180,E1 -10907.393,E2 -10907.393} C_VEL
LIN {X 0,Y 403.792,Z 679.947,A -85,B 0,C 180,E1 -10907.938,E2 -10907.938} C_VEL
LIN {X 0,Y 403.409,Z 677.864,A -85,B 0,C 180,E1 -10908.013,E2 -10908.013} C_VEL
LIN {X 0,Y 403.741,Z 670.783,A -85,B 0,C 180,E1 -10911.442,E2 -10911.442} C_VEL
LIN {X 0,Y 404.058,Z 664.291,A -85,B 0,C 180,E1 -10914.674,E2 -10914.674} C_VEL
LIN {X 0,Y 404.512,Z 656.788,A -85,B 0,C 180,E1 -10918.541,E2 -10918.541} C_VEL
LIN {X 0,Y 404.961,Z 650.843,A -85,B 0,C 180,E1 -10921.746,E2 -10921.746} C_VEL
LIN {X 0,Y 405.439,Z 645.314,A -85,B 0,C 180,E1 -10924.892,E2 -10924.892} C_VEL
LIN {X 0,Y 405.337,Z 641.696,A -85,B 0,C 180,E1 -10927.1,E2 -10927.1} C_VEL
LIN {X 0,Y 404.719,Z 637.336,A -85,B 0,C 180,E1 -10929.979,E2 -10929.979} C_VEL
LIN {X 0,Y 404.157,Z 634.146,A -85,B 0,C 180,E1 -10932.267,E2 -10932.267} C_VEL
LIN {X 0,Y 404.148,Z 634.145,A -85,B 0,C 180,E1 -10935.478,E2 -10935.478} C_VEL
LIN {X 0,Y 404.121,Z 634.15,A -85,B 0,C 180,E1 -10938.635,E2 -10938.635} C_VEL
LIN {X 0,Y 404.155,Z 634.144,A -85,B 0,C 180,E1 -10941.492,E2 -10941.492} C_VEL
LIN {X 0,Y 404.186,Z 634.14,A -85,B 0,C 180,E1 -10944.984,E2 -10944.984} C_VEL
LIN {X 0,Y 404.144,Z 634.146,A -85,B 0,C 180,E1 -10948.554,E2 -10948.554} C_VEL
LIN {X 0,Y 404.197,Z 634.137,A -85,B 0,C 180,E1 -10952,E2 -10952} C_VEL
LIN {X 0,Y 404.179,Z 634.141,A -85,B 0,C 180,E1 -10955.334,E2 -10955.334} C_VEL
LIN {X 0,Y 404.14,Z 634.146,A -85,B 0,C 180,E1 -10958.581,E2 -10958.581} C_VEL
LIN {X 0,Y 404.212,Z 634.137,A -85,B 0,C 180,E1 -10961.762,E2 -10961.762} C_VEL
LIN {X 0,Y 404.208,Z 634.137,A -85,B 0,C 180,E1 -10964.882,E2 -10964.882} C_VEL
LIN {X 0,Y 404.258,Z 634.131,A -85,B 0,C 180,E1 -10967.959,E2 -10967.959} C_VEL
LIN {X 0,Y 404.435,Z 634.106,A -85,B 0,C 180,E1 -10972.1,E2 -10972.1} C_VEL
LIN {X 0,Y 404.425,Z 634.108,A -85,B 0,C 180,E1 -10974.015,E2 -10974.015} C_VEL
LIN {X 0,Y 404.482,Z 634.104,A -85,B 0,C 180,E1 -10978.009,E2 -10978.009} C_VEL
LIN {X 0,Y 404.613,Z 634.087,A -85,B 0,C 180,E1 -10980,E2 -10980} C_VEL
LIN {X 0,Y 404.425,Z 634.112,A -85,B 0,C 180,E1 -10982.988,E2 -10982.988} C_VEL
LIN {X 0,Y 404.396,Z 634.113,A -85,B 0,C 180,E1 -10986.635,E2 -10986.635} C_VEL
LIN {X 0,Y 404.356,Z 634.17,A -85,B 0,C 180,E1 -10987.993,E2 -10987.993} C_VEL
LIN {X 0,Y 404.285,Z 637.521,A -85,B 0,C 180,E1 -10991.024,E2 -10991.024} C_VEL
LIN {X 0,Y 404.036,Z 641.073,A -85,B 0,C 180,E1 -10994.095,E2 -10994.095} C_VEL
LIN {X 0,Y 403.805,Z 644.842,A -85,B 0,C 180,E1 -10997.21,E2 -10997.21} C_VEL
LIN {X 0,Y 403.598,Z 648.776,A -85,B 0,C 180,E1 -11000.381,E2 -11000.381} C_VEL
LIN {X 0,Y 403.41,Z 652.905,A -85,B 0,C 180,E1 -11003.622,E2 -11003.622} C_VEL
LIN {X 0,Y 403.3,Z 657.387,A -85,B 0,C 180,E1 -11007.061,E2 -11007.061} C_VEL
LIN {X 0,Y 406.801,Z 672.026,A -85,B 0,C 180,E1 -11007.777,E2 -11007.777} C_VEL
LIN {X 0,Y 408.578,Z 681.788,A -85,B 0,C 180,E1 -11008.371,E2 -11008.371} C_VEL
LIN {X 0,Y 407.856,Z 693.551,A -85,B 0,C 180,E1 -11009.13,E2 -11009.13} C_VEL
LIN {X 0,Y 407.111,Z 704.526,A -85,B 0,C 180,E1 -11010.042,E2 -11010.042} C_VEL
LIN {X 0,Y 406.285,Z 714.982,A -85,B 0,C 180,E1 -11011.134,E2 -11011.134} C_VEL
LIN {X 0,Y 405.482,Z 724.36,A -85,B 0,C 180,E1 -11012.339,E2 -11012.339} C_VEL
LIN {X 0,Y 404.775,Z 733.308,A -85,B 0,C 180,E1 -11013.753,E2 -11013.753} C_VEL
LIN {X 0,Y 404.079,Z 741.562,A -85,B 0,C 180,E1 -11015.397,E2 -11015.397} C_VEL
LIN {X 0,Y 403.56,Z 748.39,A -85,B 0,C 180,E1 -11017.132,E2 -11017.132} C_VEL
LIN {X 0,Y 403.206,Z 753.54,A -85,B 0,C 180,E1 -11018.865,E2 -11018.865} C_VEL
LIN {X 0,Y 402.961,Z 757.597,A -85,B 0,C 180,E1 -11020.786,E2 -11020.786} C_VEL
LIN {X 0,Y 402.856,Z 758.727,A -85,B 0,C 180,E1 -11021.524,E2 -11021.524} C_VEL
LIN {X 0,Y 402.77,Z 760.222,A -85,B 0,C 180,E1 -11022.884,E2 -11022.884} C_VEL
LIN {X 0,Y 402.695,Z 761.005,A -85,B 0,C 180,E1 -11024.312,E2 -11024.312} C_VEL
LIN {X 0,Y 402.693,Z 760.973,A -85,B 0,C 180,E1 -11025.725,E2 -11025.725} C_VEL
LIN {X 0,Y 402.706,Z 760.123,A -85,B 0,C 180,E1 -11027.137,E2 -11027.137} C_VEL
LIN {X 0,Y 402.858,Z 758.398,A -85,B 0,C 180,E1 -11028.604,E2 -11028.604} C_VEL
LIN {X 0,Y 403.047,Z 755.697,A -85,B 0,C 180,E1 -11030.107,E2 -11030.107} C_VEL
LIN {X 0,Y 403.228,Z 751.844,A -85,B 0,C 180,E1 -11031.658,E2 -11031.658} C_VEL
LIN {X 0,Y 403.577,Z 746.714,A -85,B 0,C 180,E1 -11033.231,E2 -11033.231} C_VEL
LIN {X 0,Y 404.045,Z 740.045,A -85,B 0,C 180,E1 -11034.838,E2 -11034.838} C_VEL
LIN {X 0,Y 404.59,Z 732.815,A -85,B 0,C 180,E1 -11036.23,E2 -11036.23} C_VEL
LIN {X 0,Y 405.359,Z 723.626,A -85,B 0,C 180,E1 -11037.658,E2 -11037.658} C_VEL
LIN {X 0,Y 406.075,Z 714.175,A -85,B 0,C 180,E1 -11038.855,E2 -11038.855} C_VEL
LIN {X 0,Y 406.88,Z 703.583,A -85,B 0,C 180,E1 -11039.939,E2 -11039.939} C_VEL
LIN {X 0,Y 407.657,Z 691.32,A -85,B 0,C 180,E1 -11040.925,E2 -11040.925} C_VEL
LIN {X 0,Y 408.222,Z 681.213,A -85,B 0,C 180,E1 -11041.56,E2 -11041.56} C_VEL
LIN {X 0,Y 405.692,Z 667.942,A -85,B 0,C 180,E1 -11042.315,E2 -11042.315} C_VEL
LIN {X 0,Y 403.161,Z 656.681,A -85,B 0,C 180,E1 -11042.822,E2 -11042.822} C_VEL
LIN {X 0,Y 403.239,Z 653.325,A -85,B 0,C 180,E1 -11045.273,E2 -11045.273} C_VEL
LIN {X 0,Y 403.4,Z 648.943,A -85,B 0,C 180,E1 -11048.539,E2 -11048.539} C_VEL
LIN {X 0,Y 403.591,Z 644.724,A -85,B 0,C 180,E1 -11051.733,E2 -11051.733} C_VEL
LIN {X 0,Y 403.777,Z 640.677,A -85,B 0,C 180,E1 -11054.865,E2 -11054.865} C_VEL
LIN {X 0,Y 404.013,Z 636.768,A -85,B 0,C 180,E1 -11057.951,E2 -11057.951} C_VEL
LIN {X 0,Y 404.066,Z 634.273,A -85,B 0,C 180,E1 -11059.983,E2 -11059.983} C_VEL
LIN {X 0,Y 404.4,Z 634.114,A -85,B 0,C 180,E1 -11063.012,E2 -11063.012} C_VEL
LIN {X 0,Y 404.285,Z 634.128,A -85,B 0,C 180,E1 -11065.013,E2 -11065.013} C_VEL
LIN {X 0,Y 404.486,Z 634.098,A -85,B 0,C 180,E1 -11068.008,E2 -11068.008} C_VEL
LIN {X 0,Y 404.615,Z 634.082,A -85,B 0,C 180,E1 -11070,E2 -11070} C_VEL
LIN {X 0,Y 404.425,Z 634.111,A -85,B 0,C 180,E1 -11072.988,E2 -11072.988} C_VEL
LIN {X 0,Y 404.408,Z 634.108,A -85,B 0,C 180,E1 -11076.037,E2 -11076.037} C_VEL
LIN {X 0,Y 403.677,Z 634.204,A -85,B 0,C 180,E1 -11076.867,E2 -11076.867} C_VEL
LIN {X 0,Y 400.731,Z 634.567,A -85,B 0,C 180,E1 -11078.214,E2 -11078.214} C_VEL
LIN {X 0,Y 398.204,Z 634.883,A -85,B 0,C 180,E1 -11079.301,E2 -11079.301} C_VEL
LIN {X 0,Y 397.035,Z 635.027,A -85,B 0,C 180,E1 -11080.143,E2 -11080.143} C_VEL
LIN {X 0,Y 396.893,Z 635.045,A -85,B 0,C 180,E1 -11080.429,E2 -11080.429} C_VEL
LIN {X 0,Y 396.615,Z 635.243,A -85,B 0,C 180,E1 -11082.147,E2 -11082.147} C_VEL
LIN {X 0,Y 396.373,Z 640.228,A -85,B 0,C 180,E1 -11085.424,E2 -11085.424} C_VEL
LIN {X 0,Y 396.304,Z 643.433,A -85,B 0,C 180,E1 -11087.546,E2 -11087.546} C_VEL
LIN {X 0,Y 396.144,Z 648.332,A -85,B 0,C 180,E1 -11090.782,E2 -11090.782} C_VEL
LIN {X 0,Y 396.023,Z 653.355,A -85,B 0,C 180,E1 -11094.089,E2 -11094.089} C_VEL
LIN {X 0,Y 396,Z 656.221,A -85,B 0,C 180,E1 -11095.985,E2 -11095.985} C_VEL
LIN {X 0,Y 399.266,Z 670.955,A -85,B 0,C 180,E1 -11096.67,E2 -11096.67} C_VEL
LIN {X 0,Y 401.31,Z 682.569,A -85,B 0,C 180,E1 -11097.368,E2 -11097.368} C_VEL
LIN {X 0,Y 400.529,Z 695.028,A -85,B 0,C 180,E1 -11098.207,E2 -11098.207} C_VEL
LIN {X 0,Y 399.764,Z 705.712,A -85,B 0,C 180,E1 -11099.133,E2 -11099.133} C_VEL
LIN {X 0,Y 398.911,Z 716.515,A -85,B 0,C 180,E1 -11100.313,E2 -11100.313} C_VEL
LIN {X 0,Y 398.07,Z 726.633,A -85,B 0,C 180,E1 -11101.684,E2 -11101.684} C_VEL
LIN {X 0,Y 397.471,Z 734.14,A -85,B 0,C 180,E1 -11102.936,E2 -11102.936} C_VEL
LIN {X 0,Y 396.871,Z 741.831,A -85,B 0,C 180,E1 -11104.518,E2 -11104.518} C_VEL
LIN {X 0,Y 396.408,Z 747.996,A -85,B 0,C 180,E1 -11106.107,E2 -11106.107} C_VEL
LIN {X 0,Y 396.077,Z 752.96,A -85,B 0,C 180,E1 -11107.746,E2 -11107.746} C_VEL
LIN {X 0,Y 395.843,Z 756.186,A -85,B 0,C 180,E1 -11109.155,E2 -11109.155} C_VEL
LIN {X 0,Y 395.692,Z 758.056,A -85,B 0,C 180,E1 -11110.205,E2 -11110.205} C_VEL
LIN {X 0,Y 395.582,Z 759.961,A -85,B 0,C 180,E1 -11111.739,E2 -11111.739} C_VEL
LIN {X 0,Y 395.554,Z 760.924,A -85,B 0,C 180,E1 -11113.242,E2 -11113.242} C_VEL
LIN {X 0,Y 395.595,Z 760.816,A -85,B 0,C 180,E1 -11115.285,E2 -11115.285} C_VEL
LIN {X 0,Y 395.664,Z 759.777,A -85,B 0,C 180,E1 -11116.74,E2 -11116.74} C_VEL
LIN {X 0,Y 395.789,Z 757.858,A -85,B 0,C 180,E1 -11118.226,E2 -11118.226} C_VEL
LIN {X 0,Y 396.01,Z 754.965,A -85,B 0,C 180,E1 -11119.739,E2 -11119.739} C_VEL
LIN {X 0,Y 396.378,Z 749.846,A -85,B 0,C 180,E1 -11121.642,E2 -11121.642} C_VEL
LIN {X 0,Y 396.82,Z 743.975,A -85,B 0,C 180,E1 -11123.292,E2 -11123.292} C_VEL
LIN {X 0,Y 397.48,Z 736.066,A -85,B 0,C 180,E1 -11125.014,E2 -11125.014} C_VEL
LIN {X 0,Y 398.294,Z 727.639,A -85,B 0,C 180,E1 -11126.478,E2 -11126.478} C_VEL
LIN {X 0,Y 399.042,Z 718.917,A -85,B 0,C 180,E1 -11127.712,E2 -11127.712} C_VEL
LIN {X 0,Y 399.95,Z 708.289,A -85,B 0,C 180,E1 -11128.924,E2 -11128.924} C_VEL
LIN {X 0,Y 400.7,Z 698.109,A -85,B 0,C 180,E1 -11129.863,E2 -11129.863} C_VEL
LIN {X 0,Y 401.551,Z 686.105,A -85,B 0,C 180,E1 -11130.734,E2 -11130.734} C_VEL
LIN {X 0,Y 401.636,Z 682.163,A -85,B 0,C 180,E1 -11130.978,E2 -11130.978} C_VEL
LIN {X 0,Y 399.43,Z 670.304,A -85,B 0,C 180,E1 -11131.703,E2 -11131.703} C_VEL
LIN {X 0,Y 396.098,Z 656.735,A -85,B 0,C 180,E1 -11132.376,E2 -11132.376} C_VEL
LIN {X 0,Y 396.208,Z 653.021,A -85,B 0,C 180,E1 -11134.804,E2 -11134.804} C_VEL
LIN {X 0,Y 396.244,Z 647.883,A -85,B 0,C 180,E1 -11138.132,E2 -11138.132} C_VEL
LIN {X 0,Y 396.395,Z 642.893,A -85,B 0,C 180,E1 -11141.389,E2 -11141.389} C_VEL
LIN {X 0,Y 396.511,Z 637.707,A -85,B 0,C 180,E1 -11144.581,E2 -11144.581} C_VEL
LIN {X 0,Y 396.709,Z 635.077,A -85,B 0,C 180,E1 -11146.293,E2 -11146.293} C_VEL
LIN {X 0,Y 397.021,Z 635.034,A -85,B 0,C 180,E1 -11148.772,E2 -11148.772} C_VEL
LIN {X 0,Y 397.362,Z 634.992,A -85,B 0,C 180,E1 -11152.07,E2 -11152.07} C_VEL
LIN {X 0,Y 397.253,Z 635.005,A -85,B 0,C 180,E1 -11154.925,E2 -11154.925} C_VEL
LIN {X 0,Y 397.448,Z 634.979,A -85,B 0,C 180,E1 -11157.973,E2 -11157.973} C_VEL
LIN {X 0,Y 397.579,Z 634.963,A -85,B 0,C 180,E1 -11160,E2 -11160} C_VEL
LIN {X 0,Y 397.379,Z 634.988,A -85,B 0,C 180,E1 -11163.041,E2 -11163.041} C_VEL
LIN {X 0,Y 397.36,Z 634.99,A -85,B 0,C 180,E1 -11167.112,E2 -11167.112} C_VEL
LIN {X 0,Y 397.215,Z 635.007,A -85,B 0,C 180,E1 -11170.191,E2 -11170.191} C_VEL
LIN {X 0,Y 397.222,Z 635.007,A -85,B 0,C 180,E1 -11173.321,E2 -11173.321} C_VEL
LIN {X 0,Y 397.178,Z 635.012,A -85,B 0,C 180,E1 -11177.155,E2 -11177.155} C_VEL
LIN {X 0,Y 397.099,Z 635.023,A -85,B 0,C 180,E1 -11180.73,E2 -11180.73} C_VEL
LIN {X 0,Y 397.129,Z 635.017,A -85,B 0,C 180,E1 -11184.019,E2 -11184.019} C_VEL
LIN {X 0,Y 397.191,Z 635.011,A -85,B 0,C 180,E1 -11187.39,E2 -11187.39} C_VEL
LIN {X 0,Y 397.082,Z 635.023,A -85,B 0,C 180,E1 -11190.882,E2 -11190.882} C_VEL
LIN {X 0,Y 397.123,Z 635.02,A -85,B 0,C 180,E1 -11194.494,E2 -11194.494} C_VEL
LIN {X 0,Y 397.103,Z 635.021,A -85,B 0,C 180,E1 -11198.275,E2 -11198.275} C_VEL
LIN {X 0,Y 397.086,Z 635.024,A -85,B 0,C 180,E1 -11200.909,E2 -11200.909} C_VEL
LIN {X 0,Y 397.099,Z 635.023,A -85,B 0,C 180,E1 -11203.649,E2 -11203.649} C_VEL
LIN {X 0,Y 397.1,Z 635.023,A -85,B 0,C 180,E1 -11206.522,E2 -11206.522} C_VEL
LIN {X 0,Y 397.152,Z 635.181,A -85,B 0,C 180,E1 -11208.764,E2 -11208.764} C_VEL
LIN {X 0,Y 397.979,Z 640.147,A -85,B 0,C 180,E1 -11211.825,E2 -11211.825} C_VEL
LIN {X 0,Y 398.405,Z 644.539,A -85,B 0,C 180,E1 -11214.4,E2 -11214.4} C_VEL
LIN {X 0,Y 398.044,Z 650.002,A -85,B 0,C 180,E1 -11217.418,E2 -11217.418} C_VEL
LIN {X 0,Y 397.569,Z 656.563,A -85,B 0,C 180,E1 -11220.914,E2 -11220.914} C_VEL
LIN {X 0,Y 397.074,Z 663.504,A -85,B 0,C 180,E1 -11224.512,E2 -11224.512} C_VEL
LIN {X 0,Y 396.687,Z 670.741,A -85,B 0,C 180,E1 -11228.158,E2 -11228.158} C_VEL
LIN {X 0,Y 396.369,Z 678.325,A -85,B 0,C 180,E1 -11231.891,E2 -11231.891} C_VEL
LIN {X 0,Y 399.075,Z 693.586,A -85,B 0,C 180,E1 -11232.551,E2 -11232.551} C_VEL
LIN {X 0,Y 400.742,Z 706.523,A -85,B 0,C 180,E1 -11233.292,E2 -11233.292} C_VEL
LIN {X 0,Y 400.517,Z 714.571,A -85,B 0,C 180,E1 -11233.826,E2 -11233.826} C_VEL
LIN {X 0,Y 399.703,Z 725.587,A -85,B 0,C 180,E1 -11234.708,E2 -11234.708} C_VEL
LIN {X 0,Y 398.952,Z 735.736,A -85,B 0,C 180,E1 -11235.723,E2 -11235.723} C_VEL
LIN {X 0,Y 398.17,Z 746.008,A -85,B 0,C 180,E1 -11236.995,E2 -11236.995} C_VEL
LIN {X 0,Y 397.313,Z 755.861,A -85,B 0,C 180,E1 -11238.522,E2 -11238.522} C_VEL
LIN {X 0,Y 396.698,Z 763.779,A -85,B 0,C 180,E1 -11240.054,E2 -11240.054} C_VEL
LIN {X 0,Y 396.349,Z 769.146,A -85,B 0,C 180,E1 -11241.332,E2 -11241.332} C_VEL
LIN {X 0,Y 396.01,Z 774.386,A -85,B 0,C 180,E1 -11242.864,E2 -11242.864} C_VEL
LIN {X 0,Y 395.856,Z 777.852,A -85,B 0,C 180,E1 -11244.153,E2 -11244.153} C_VEL
LIN {X 0,Y 395.782,Z 781.446,A -85,B 0,C 180,E1 -11245.927,E2 -11245.927} C_VEL
LIN {X 0,Y 395.725,Z 782.897,A -85,B 0,C 180,E1 -11246.946,E2 -11246.946} C_VEL
LIN {X 0,Y 395.76,Z 783.919,A -85,B 0,C 180,E1 -11247.965,E2 -11247.965} C_VEL
LIN {X 0,Y 395.79,Z 784.546,A -85,B 0,C 180,E1 -11248.983,E2 -11248.983} C_VEL
LIN {X 0,Y 395.778,Z 784.782,A -85,B 0,C 180,E1 -11250,E2 -11250} C_VEL
LIN {X 0,Y 395.79,Z 784.591,A -85,B 0,C 180,E1 -11251.018,E2 -11251.018} C_VEL
LIN {X 0,Y 395.759,Z 783.984,A -85,B 0,C 180,E1 -11252.036,E2 -11252.036} C_VEL
LIN {X 0,Y 395.783,Z 781.587,A -85,B 0,C 180,E1 -11254.073,E2 -11254.073} C_VEL
LIN {X 0,Y 395.853,Z 778.639,A -85,B 0,C 180,E1 -11255.604,E2 -11255.604} C_VEL
LIN {X 0,Y 396.057,Z 774.652,A -85,B 0,C 180,E1 -11257.136,E2 -11257.136} C_VEL
LIN {X 0,Y 396.4,Z 768.534,A -85,B 0,C 180,E1 -11258.925,E2 -11258.925} C_VEL
LIN {X 0,Y 396.92,Z 761.842,A -85,B 0,C 180,E1 -11260.457,E2 -11260.457} C_VEL
LIN {X 0,Y 397.62,Z 753.565,A -85,B 0,C 180,E1 -11261.987,E2 -11261.987} C_VEL
LIN {X 0,Y 398.405,Z 745.12,A -85,B 0,C 180,E1 -11263.258,E2 -11263.258} C_VEL
LIN {X 0,Y 399.134,Z 734.964,A -85,B 0,C 180,E1 -11264.506,E2 -11264.506} C_VEL
LIN {X 0,Y 400.102,Z 723.084,A -85,B 0,C 180,E1 -11265.669,E2 -11265.669} C_VEL
LIN {X 0,Y 400.941,Z 711.951,A -85,B 0,C 180,E1 -11266.525,E2 -11266.525} C_VEL
LIN {X 0,Y 401.021,Z 706.615,A -85,B 0,C 180,E1 -11266.877,E2 -11266.877} C_VEL
LIN {X 0,Y 399.359,Z 693.179,A -85,B 0,C 180,E1 -11267.671,E2 -11267.671} C_VEL
LIN {X 0,Y 396.85,Z 680.114,A -85,B 0,C 180,E1 -11268.277,E2 -11268.277} C_VEL
LIN {X 0,Y 396.364,Z 677.596,A -85,B 0,C 180,E1 -11268.395,E2 -11268.395} C_VEL
LIN {X 0,Y 396.71,Z 670.641,A -85,B 0,C 180,E1 -11271.841,E2 -11271.841} C_VEL
LIN {X 0,Y 397.078,Z 663.502,A -85,B 0,C 180,E1 -11275.489,E2 -11275.489} C_VEL
LIN {X 0,Y 397.484,Z 657.789,A -85,B 0,C 180,E1 -11278.516,E2 -11278.516} C_VEL
LIN {X 0,Y 397.976,Z 651.404,A -85,B 0,C 180,E1 -11282.043,E2 -11282.043} C_VEL
LIN {X 0,Y 398.434,Z 646.349,A -85,B 0,C 180,E1 -11284.979,E2 -11284.979} C_VEL
LIN {X 0,Y 398.28,Z 642.434,A -85,B 0,C 180,E1 -11287.433,E2 -11287.433} C_VEL
LIN {X 0,Y 397.605,Z 637.889,A -85,B 0,C 180,E1 -11290.53,E2 -11290.53} C_VEL
LIN {X 0,Y 397.099,Z 635.025,A -85,B 0,C 180,E1 -11292.779,E2 -11292.779} C_VEL
LIN {X 0,Y 397.104,Z 635.023,A -85,B 0,C 180,E1 -11296.521,E2 -11296.521} C_VEL
LIN {X 0,Y 397.115,Z 635.022,A -85,B 0,C 180,E1 -11300.423,E2 -11300.423} C_VEL
LIN {X 0,Y 397.11,Z 635.021,A -85,B 0,C 180,E1 -11304.265,E2 -11304.265} C_VEL
LIN {X 0,Y 397.116,Z 635.021,A -85,B 0,C 180,E1 -11306.727,E2 -11306.727} C_VEL
LIN {X 0,Y 397.126,Z 635.019,A -85,B 0,C 180,E1 -11310.296,E2 -11310.296} C_VEL
LIN {X 0,Y 397.196,Z 635.011,A -85,B 0,C 180,E1 -11312.61,E2 -11312.61} C_VEL
LIN {X 0,Y 397.135,Z 635.015,A -85,B 0,C 180,E1 -11315.982,E2 -11315.982} C_VEL
LIN {X 0,Y 397.14,Z 635.018,A -85,B 0,C 180,E1 -11319.705,E2 -11319.705} C_VEL
LIN {X 0,Y 397.183,Z 635.013,A -85,B 0,C 180,E1 -11322.845,E2 -11322.845} C_VEL
LIN {X 0,Y 397.23,Z 635.007,A -85,B 0,C 180,E1 -11326.703,E2 -11326.703} C_VEL
LIN {X 0,Y 397.22,Z 635.005,A -85,B 0,C 180,E1 -11329.809,E2 -11329.809} C_VEL
LIN {X 0,Y 397.366,Z 634.99,A -85,B 0,C 180,E1 -11332.888,E2 -11332.888} C_VEL
LIN {X 0,Y 397.257,Z 635.004,A -85,B 0,C 180,E1 -11334.925,E2 -11334.925} C_VEL
LIN {X 0,Y 397.451,Z 634.98,A -85,B 0,C 180,E1 -11337.973,E2 -11337.973} C_VEL
LIN {X 0,Y 397.582,Z 634.963,A -85,B 0,C 180,E1 -11340,E2 -11340} C_VEL
LIN {X 0,Y 397.384,Z 634.989,A -85,B 0,C 180,E1 -11343.041,E2 -11343.041} C_VEL
LIN {X 0,Y 397.345,Z 634.991,A -85,B 0,C 180,E1 -11346.632,E2 -11346.632} C_VEL
LIN {X 0,Y 397.363,Z 635.434,A -85,B 0,C 180,E1 -11348.134,E2 -11348.134} C_VEL
LIN {X 0,Y 397.24,Z 638.817,A -85,B 0,C 180,E1 -11351.222,E2 -11351.222} C_VEL
LIN {X 0,Y 396.98,Z 642.371,A -85,B 0,C 180,E1 -11354.351,E2 -11354.351} C_VEL
LIN {X 0,Y 396.739,Z 646.141,A -85,B 0,C 180,E1 -11357.526,E2 -11357.526} C_VEL
LIN {X 0,Y 396.524,Z 650.092,A -85,B 0,C 180,E1 -11360.762,E2 -11360.762} C_VEL
LIN {X 0,Y 396.348,Z 654.255,A -85,B 0,C 180,E1 -11364.069,E2 -11364.069} C_VEL
LIN {X 0,Y 396.243,Z 657.786,A -85,B 0,C 180,E1 -11366.713,E2 -11366.713} C_VEL
LIN {X 0,Y 399.73,Z 671.739,A -85,B 0,C 180,E1 -11367.414,E2 -11367.414} C_VEL
LIN {X 0,Y 401.801,Z 682.835,A -85,B 0,C 180,E1 -11368.108,E2 -11368.108} C_VEL
LIN {X 0,Y 401.051,Z 694.542,A -85,B 0,C 180,E1 -11368.889,E2 -11368.889} C_VEL
LIN {X 0,Y 400.311,Z 704.488,A -85,B 0,C 180,E1 -11369.734,E2 -11369.734} C_VEL
LIN {X 0,Y 399.459,Z 714.84,A -85,B 0,C 180,E1 -11370.825,E2 -11370.825} C_VEL
LIN {X 0,Y 398.53,Z 725.107,A -85,B 0,C 180,E1 -11372.17,E2 -11372.17} C_VEL
LIN {X 0,Y 397.845,Z 733.388,A -85,B 0,C 180,E1 -11373.51,E2 -11373.51} C_VEL
LIN {X 0,Y 397.176,Z 740.75,A -85,B 0,C 180,E1 -11374.971,E2 -11374.971} C_VEL
LIN {X 0,Y 396.552,Z 747.773,A -85,B 0,C 180,E1 -11376.737,E2 -11376.737} C_VEL
LIN {X 0,Y 396.2,Z 752.821,A -85,B 0,C 180,E1 -11378.378,E2 -11378.378} C_VEL
LIN {X 0,Y 395.933,Z 757.037,A -85,B 0,C 180,E1 -11380.246,E2 -11380.246} C_VEL
LIN {X 0,Y 395.749,Z 759.378,A -85,B 0,C 180,E1 -11381.766,E2 -11381.766} C_VEL
LIN {X 0,Y 395.62,Z 761.063,A -85,B 0,C 180,E1 -11383.854,E2 -11383.854} C_VEL
LIN {X 0,Y 395.592,Z 761.26,A -85,B 0,C 180,E1 -11385.287,E2 -11385.287} C_VEL
LIN {X 0,Y 395.587,Z 760.657,A -85,B 0,C 180,E1 -11386.753,E2 -11386.753} C_VEL
LIN {X 0,Y 395.727,Z 759.194,A -85,B 0,C 180,E1 -11388.237,E2 -11388.237} C_VEL
LIN {X 0,Y 395.926,Z 756.77,A -85,B 0,C 180,E1 -11389.755,E2 -11389.755} C_VEL
LIN {X 0,Y 396.159,Z 752.44,A -85,B 0,C 180,E1 -11391.617,E2 -11391.617} C_VEL
LIN {X 0,Y 396.505,Z 747.272,A -85,B 0,C 180,E1 -11393.258,E2 -11393.258} C_VEL
LIN {X 0,Y 396.964,Z 741.124,A -85,B 0,C 180,E1 -11394.792,E2 -11394.792} C_VEL
LIN {X 0,Y 397.523,Z 734.179,A -85,B 0,C 180,E1 -11396.195,E2 -11396.195} C_VEL
LIN {X 0,Y 398.268,Z 725.232,A -85,B 0,C 180,E1 -11397.66,E2 -11397.66} C_VEL
LIN {X 0,Y 399.11,Z 715.036,A -85,B 0,C 180,E1 -11398.998,E2 -11398.998} C_VEL
LIN {X 0,Y 399.942,Z 704.711,A -85,B 0,C 180,E1 -11400.091,E2 -11400.091} C_VEL
LIN {X 0,Y 400.684,Z 693.558,A -85,B 0,C 180,E1 -11401.034,E2 -11401.034} C_VEL
LIN {X 0,Y 401.342,Z 682.2,A -85,B 0,C 180,E1 -11401.783,E2 -11401.783} C_VEL
LIN {X 0,Y 398.846,Z 668.971,A -85,B 0,C 180,E1 -11402.564,E2 -11402.564} C_VEL
LIN {X 0,Y 396.098,Z 656.935,A -85,B 0,C 180,E1 -11403.099,E2 -11403.099} C_VEL
LIN {X 0,Y 396.178,Z 653.109,A -85,B 0,C 180,E1 -11405.92,E2 -11405.92} C_VEL
LIN {X 0,Y 396.384,Z 648.73,A -85,B 0,C 180,E1 -11409.23,E2 -11409.23} C_VEL
LIN {X 0,Y 396.572,Z 644.546,A -85,B 0,C 180,E1 -11412.466,E2 -11412.466} C_VEL
LIN {X 0,Y 396.799,Z 640.516,A -85,B 0,C 180,E1 -11415.643,E2 -11415.643} C_VEL
LIN {X 0,Y 396.964,Z 637.904,A -85,B 0,C 180,E1 -11417.734,E2 -11417.734} C_VEL
LIN {X 0,Y 397.019,Z 635.391,A -85,B 0,C 180,E1 -11419.803,E2 -11419.803} C_VEL
LIN {X 0,Y 397.278,Z 634.996,A -85,B 0,C 180,E1 -11421.864,E2 -11421.864} C_VEL
LIN {X 0,Y 397.375,Z 634.984,A -85,B 0,C 180,E1 -11423.908,E2 -11423.908} C_VEL
LIN {X 0,Y 397.455,Z 634.974,A -85,B 0,C 180,E1 -11427.973,E2 -11427.973} C_VEL
LIN {X 0,Y 397.585,Z 634.958,A -85,B 0,C 180,E1 -11430,E2 -11430} C_VEL
LIN {X 0,Y 397.384,Z 634.987,A -85,B 0,C 180,E1 -11433.041,E2 -11433.041} C_VEL
LIN {X 0,Y 397.362,Z 634.986,A -85,B 0,C 180,E1 -11436.091,E2 -11436.091} C_VEL
LIN {X 0,Y 397.231,Z 635.003,A -85,B 0,C 180,E1 -11438.136,E2 -11438.136} C_VEL
LIN {X 0,Y 396.893,Z 635.045,A -85,B 0,C 180,E1 -11440.429,E2 -11440.429} C_VEL
LIN {X 0,Y 396.067,Z 635.338,A -85,B 0,C 180,E1 -11441.271,E2 -11441.271} C_VEL
LIN {X 0,Y 393.046,Z 636.728,A -85,B 0,C 180,E1 -11442.626,E2 -11442.626} C_VEL
LIN {X 0,Y 390.541,Z 638.336,A -85,B 0,C 180,E1 -11443.713,E2 -11443.713} C_VEL
LIN {X 0,Y 389.444,Z 639.65,A -85,B 0,C 180,E1 -11444.552,E2 -11444.552} C_VEL
LIN {X 0,Y 389.338,Z 640.085,A -85,B 0,C 180,E1 -11444.837,E2 -11444.837} C_VEL
LIN {X 0,Y 389.222,Z 644.666,A -85,B 0,C 180,E1 -11447.876,E2 -11447.876} C_VEL
LIN {X 0,Y 389.052,Z 649.627,A -85,B 0,C 180,E1 -11451.179,E2 -11451.179} C_VEL
LIN {X 0,Y 388.936,Z 654.674,A -85,B 0,C 180,E1 -11454.557,E2 -11454.557} C_VEL
LIN {X 0,Y 388.947,Z 656.409,A -85,B 0,C 180,E1 -11455.7,E2 -11455.7} C_VEL
LIN {X 0,Y 392.058,Z 670.417,A -85,B 0,C 180,E1 -11456.337,E2 -11456.337} C_VEL
LIN {X 0,Y 394.364,Z 683.057,A -85,B 0,C 180,E1 -11457.11,E2 -11457.11} C_VEL
LIN {X 0,Y 393.66,Z 695.169,A -85,B 0,C 180,E1 -11457.945,E2 -11457.945} C_VEL
LIN {X 0,Y 392.876,Z 705.798,A -85,B 0,C 180,E1 -11458.88,E2 -11458.88} C_VEL
LIN {X 0,Y 391.939,Z 717.084,A -85,B 0,C 180,E1 -11460.137,E2 -11460.137} C_VEL
LIN {X 0,Y 391.158,Z 726.269,A -85,B 0,C 180,E1 -11461.402,E2 -11461.402} C_VEL
LIN {X 0,Y 390.508,Z 733.891,A -85,B 0,C 180,E1 -11462.677,E2 -11462.677} C_VEL
LIN {X 0,Y 389.868,Z 741.677,A -85,B 0,C 180,E1 -11464.285,E2 -11464.285} C_VEL
LIN {X 0,Y 389.321,Z 748.589,A -85,B 0,C 180,E1 -11466.1,E2 -11466.1} C_VEL
LIN {X 0,Y 388.974,Z 753.767,A -85,B 0,C 180,E1 -11467.901,E2 -11467.901} C_VEL
LIN {X 0,Y 388.646,Z 757.853,A -85,B 0,C 180,E1 -11469.908,E2 -11469.908} C_VEL
LIN {X 0,Y 388.496,Z 760.392,A -85,B 0,C 180,E1 -11472.015,E2 -11472.015} C_VEL
LIN {X 0,Y 388.487,Z 761.209,A -85,B 0,C 180,E1 -11473.645,E2 -11473.645} C_VEL
LIN {X 0,Y 388.507,Z 761.101,A -85,B 0,C 180,E1 -11475.13,E2 -11475.13} C_VEL
LIN {X 0,Y 388.575,Z 760.205,A -85,B 0,C 180,E1 -11476.584,E2 -11476.584} C_VEL
LIN {X 0,Y 388.679,Z 758.524,A -85,B 0,C 180,E1 -11478.008,E2 -11478.008} C_VEL
LIN {X 0,Y 388.989,Z 754.604,A -85,B 0,C 180,E1 -11480.104,E2 -11480.104} C_VEL
LIN {X 0,Y 389.301,Z 750.807,A -85,B 0,C 180,E1 -11481.552,E2 -11481.552} C_VEL
LIN {X 0,Y 389.651,Z 745.944,A -85,B 0,C 180,E1 -11483.016,E2 -11483.016} C_VEL
LIN {X 0,Y 390.242,Z 739.82,A -85,B 0,C 180,E1 -11484.496,E2 -11484.496} C_VEL
LIN {X 0,Y 390.972,Z 731.412,A -85,B 0,C 180,E1 -11486.134,E2 -11486.134} C_VEL
LIN {X 0,Y 391.887,Z 722.267,A -85,B 0,C 180,E1 -11487.549,E2 -11487.549} C_VEL
LIN {X 0,Y 392.856,Z 711.739,A -85,B 0,C 180,E1 -11488.861,E2 -11488.861} C_VEL
LIN {X 0,Y 393.663,Z 701.752,A -85,B 0,C 180,E1 -11489.867,E2 -11489.867} C_VEL
LIN {X 0,Y 394.527,Z 690.108,A -85,B 0,C 180,E1 -11490.793,E2 -11490.793} C_VEL
LIN {X 0,Y 394.914,Z 684.857,A -85,B 0,C 180,E1 -11491.136,E2 -11491.136} C_VEL
LIN {X 0,Y 393.327,Z 674.746,A -85,B 0,C 180,E1 -11491.804,E2 -11491.804} C_VEL
LIN {X 0,Y 390.327,Z 661.74,A -85,B 0,C 180,E1 -11492.515,E2 -11492.515} C_VEL
LIN {X 0,Y 389.054,Z 656.911,A -85,B 0,C 180,E1 -11492.761,E2 -11492.761} C_VEL
LIN {X 0,Y 389.122,Z 652.809,A -85,B 0,C 180,E1 -11495.455,E2 -11495.455} C_VEL
LIN {X 0,Y 389.228,Z 647.659,A -85,B 0,C 180,E1 -11498.831,E2 -11498.831} C_VEL
LIN {X 0,Y 389.357,Z 642.5,A -85,B 0,C 180,E1 -11502.13,E2 -11502.13} C_VEL
LIN {X 0,Y 389.651,Z 636.204,A -85,B 0,C 180,E1 -11506.173,E2 -11506.173} C_VEL
LIN {X 0,Y 389.776,Z 635.941,A -85,B 0,C 180,E1 -11506.819,E2 -11506.819} C_VEL
LIN {X 0,Y 390.075,Z 635.898,A -85,B 0,C 180,E1 -11509.62,E2 -11509.62} C_VEL
LIN {X 0,Y 390.298,Z 635.872,A -85,B 0,C 180,E1 -11512.759,E2 -11512.759} C_VEL
LIN {X 0,Y 390.225,Z 635.88,A -85,B 0,C 180,E1 -11514.833,E2 -11514.833} C_VEL
LIN {X 0,Y 390.417,Z 635.855,A -85,B 0,C 180,E1 -11517.937,E2 -11517.937} C_VEL
LIN {X 0,Y 390.548,Z 635.839,A -85,B 0,C 180,E1 -11520,E2 -11520} C_VEL
LIN {X 0,Y 390.313,Z 635.869,A -85,B 0,C 180,E1 -11523.096,E2 -11523.096} C_VEL
LIN {X 0,Y 390.326,Z 635.866,A -85,B 0,C 180,E1 -11526.202,E2 -11526.202} C_VEL
LIN {X 0,Y 390.31,Z 635.868,A -85,B 0,C 180,E1 -11528.282,E2 -11528.282} C_VEL
LIN {X 0,Y 390.167,Z 635.885,A -85,B 0,C 180,E1 -11532.483,E2 -11532.483} C_VEL
LIN {X 0,Y 390.135,Z 635.891,A -85,B 0,C 180,E1 -11535.677,E2 -11535.677} C_VEL
LIN {X 0,Y 390.102,Z 635.892,A -85,B 0,C 180,E1 -11538.922,E2 -11538.922} C_VEL
LIN {X 0,Y 390.036,Z 635.902,A -85,B 0,C 180,E1 -11542.234,E2 -11542.234} C_VEL
LIN {X 0,Y 390.116,Z 635.892,A -85,B 0,C 180,E1 -11545.744,E2 -11545.744} C_VEL
LIN {X 0,Y 390.062,Z 635.898,A -85,B 0,C 180,E1 -11549.109,E2 -11549.109} C_VEL
LIN {X 0,Y 390.041,Z 635.901,A -85,B 0,C 180,E1 -11552.722,E2 -11552.722} C_VEL
LIN {X 0,Y 390.054,Z 635.898,A -85,B 0,C 180,E1 -11555.826,E2 -11555.826} C_VEL
LIN {X 0,Y 390.069,Z 635.899,A -85,B 0,C 180,E1 -11559.219,E2 -11559.219} C_VEL
LIN {X 0,Y 390.04,Z 635.901,A -85,B 0,C 180,E1 -11562.375,E2 -11562.375} C_VEL
LIN {X 0,Y 390.042,Z 635.902,A -85,B 0,C 180,E1 -11565.355,E2 -11565.355} C_VEL
LIN {X 0,Y 390.074,Z 635.927,A -85,B 0,C 180,E1 -11568.449,E2 -11568.449} C_VEL
LIN {X 0,Y 390.957,Z 641.034,A -85,B 0,C 180,E1 -11571.672,E2 -11571.672} C_VEL
LIN {X 0,Y 391.35,Z 644.778,A -85,B 0,C 180,E1 -11573.914,E2 -11573.914} C_VEL
LIN {X 0,Y 391.145,Z 649.804,A -85,B 0,C 180,E1 -11576.77,E2 -11576.77} C_VEL
LIN {X 0,Y 390.527,Z 657.436,A -85,B 0,C 180,E1 -11580.929,E2 -11580.929} C_VEL
LIN {X 0,Y 390.022,Z 663.975,A -85,B 0,C 180,E1 -11584.376,E2 -11584.376} C_VEL
LIN {X 0,Y 389.682,Z 670.525,A -85,B 0,C 180,E1 -11587.745,E2 -11587.745} C_VEL
LIN {X 0,Y 389.305,Z 677.051,A -85,B 0,C 180,E1 -11591.038,E2 -11591.038} C_VEL
LIN {X 0,Y 389.317,Z 678.324,A -85,B 0,C 180,E1 -11591.604,E2 -11591.604} C_VEL
LIN {X 0,Y 391.804,Z 692.161,A -85,B 0,C 180,E1 -11592.187,E2 -11592.187} C_VEL
LIN {X 0,Y 393.527,Z 704.872,A -85,B 0,C 180,E1 -11592.914,E2 -11592.914} C_VEL
LIN {X 0,Y 393.899,Z 710.888,A -85,B 0,C 180,E1 -11593.317,E2 -11593.317} C_VEL
LIN {X 0,Y 393.032,Z 722.274,A -85,B 0,C 180,E1 -11594.176,E2 -11594.176} C_VEL
LIN {X 0,Y 392.237,Z 732.982,A -85,B 0,C 180,E1 -11595.208,E2 -11595.208} C_VEL
LIN {X 0,Y 391.322,Z 743.736,A -85,B 0,C 180,E1 -11596.499,E2 -11596.499} C_VEL
LIN {X 0,Y 390.596,Z 752.491,A -85,B 0,C 180,E1 -11597.795,E2 -11597.795} C_VEL
LIN {X 0,Y 389.869,Z 761.003,A -85,B 0,C 180,E1 -11599.353,E2 -11599.353} C_VEL
LIN {X 0,Y 389.376,Z 767.838,A -85,B 0,C 180,E1 -11600.914,E2 -11600.914} C_VEL
LIN {X 0,Y 388.94,Z 774.113,A -85,B 0,C 180,E1 -11602.734,E2 -11602.734} C_VEL
LIN {X 0,Y 388.755,Z 777.977,A -85,B 0,C 180,E1 -11604.205,E2 -11604.205} C_VEL
LIN {X 0,Y 388.707,Z 781.203,A -85,B 0,C 180,E1 -11605.853,E2 -11605.853} C_VEL
LIN {X 0,Y 388.633,Z 782.666,A -85,B 0,C 180,E1 -11606.891,E2 -11606.891} C_VEL
LIN {X 0,Y 388.659,Z 783.693,A -85,B 0,C 180,E1 -11607.928,E2 -11607.928} C_VEL
LIN {X 0,Y 388.702,Z 784.327,A -85,B 0,C 180,E1 -11608.964,E2 -11608.964} C_VEL
LIN {X 0,Y 388.707,Z 784.568,A -85,B 0,C 180,E1 -11610,E2 -11610} C_VEL
LIN {X 0,Y 388.702,Z 784.387,A -85,B 0,C 180,E1 -11611.036,E2 -11611.036} C_VEL
LIN {X 0,Y 388.658,Z 783.783,A -85,B 0,C 180,E1 -11612.073,E2 -11612.073} C_VEL
LIN {X 0,Y 388.708,Z 781.394,A -85,B 0,C 180,E1 -11614.148,E2 -11614.148} C_VEL
LIN {X 0,Y 388.774,Z 778.211,A -85,B 0,C 180,E1 -11615.822,E2 -11615.822} C_VEL
LIN {X 0,Y 388.975,Z 774.484,A -85,B 0,C 180,E1 -11617.266,E2 -11617.266} C_VEL
LIN {X 0,Y 389.369,Z 768.393,A -85,B 0,C 180,E1 -11619.087,E2 -11619.087} C_VEL
LIN {X 0,Y 389.887,Z 761.726,A -85,B 0,C 180,E1 -11620.648,E2 -11620.648} C_VEL
LIN {X 0,Y 390.651,Z 753.468,A -85,B 0,C 180,E1 -11622.204,E2 -11622.204} C_VEL
LIN {X 0,Y 391.466,Z 745.047,A -85,B 0,C 180,E1 -11623.497,E2 -11623.497} C_VEL
LIN {X 0,Y 392.249,Z 734.934,A -85,B 0,C 180,E1 -11624.766,E2 -11624.766} C_VEL
LIN {X 0,Y 393.267,Z 723.097,A -85,B 0,C 180,E1 -11625.948,E2 -11625.948} C_VEL
LIN {X 0,Y 394.149,Z 712.135,A -85,B 0,C 180,E1 -11626.811,E2 -11626.811} C_VEL
LIN {X 0,Y 394.137,Z 707.017,A -85,B 0,C 180,E1 -11627.164,E2 -11627.164} C_VEL
LIN {X 0,Y 392.507,Z 693.856,A -85,B 0,C 180,E1 -11627.977,E2 -11627.977} C_VEL
LIN {X 0,Y 390.172,Z 681.677,A -85,B 0,C 180,E1 -11628.578,E2 -11628.578} C_VEL
LIN {X 0,Y 389.304,Z 677.379,A -85,B 0,C 180,E1 -11628.771,E2 -11628.771} C_VEL
LIN {X 0,Y 389.69,Z 670.508,A -85,B 0,C 180,E1 -11632.255,E2 -11632.255} C_VEL
LIN {X 0,Y 390.052,Z 663.89,A -85,B 0,C 180,E1 -11635.722,E2 -11635.722} C_VEL
LIN {X 0,Y 390.493,Z 657.716,A -85,B 0,C 180,E1 -11639.074,E2 -11639.074} C_VEL
LIN {X 0,Y 391.043,Z 651.452,A -85,B 0,C 180,E1 -11642.628,E2 -11642.628} C_VEL
LIN {X 0,Y 391.447,Z 647.373,A -85,B 0,C 180,E1 -11645.067,E2 -11645.067} C_VEL
LIN {X 0,Y 391.231,Z 643.171,A -85,B 0,C 180,E1 -11647.776,E2 -11647.776} C_VEL
LIN {X 0,Y 390.549,Z 638.74,A -85,B 0,C 180,E1 -11650.905,E2 -11650.905} C_VEL
LIN {X 0,Y 390.083,Z 635.898,A -85,B 0,C 180,E1 -11653.207,E2 -11653.207} C_VEL
LIN {X 0,Y 390.059,Z 635.9,A -85,B 0,C 180,E1 -11656.79,E2 -11656.79} C_VEL
LIN {X 0,Y 390.058,Z 635.903,A -85,B 0,C 180,E1 -11659.561,E2 -11659.561} C_VEL
